KUKA KRL program: EPS_2_25618_SANMH09_A_20250918115516.src

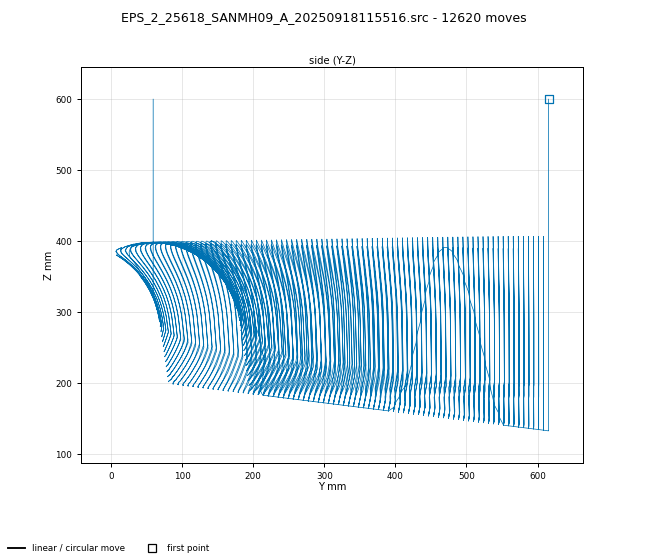
[picture p0: tool path of EPS_2_25618_SANMH09_A_20250918115516.src, 12620 of 12622 moves have a stored position in this frame; points joined in program order, loops and branches not executed]
&ACCESS RVP
&REL 4
&COMMENT QRS 19112012
&PARAM EDITMASK = *
DEF PART()
EXT BAS (BAS_COMMAND :IN,REAL :IN )
INT I
BAS (#INITMOV,0 )

;KUKA QRS Post kuka4.cps  Date:22-06-2017 !

File_ID=2845

QRS_PRE_INIT()

;Init var - Until changes are made in qrs_pre_init
Outlet_Square_prg=0
Inlet_1_Square_prg=0
Inlet_2_Square_prg=0
Inlet_3_Square_prg=0
Inlet_4_Square_prg=0
Inlet_5_Square_prg=0

Outlet_1={X 0.000, Y 546.330, Z 306.500, B 0.000, E1 0.000 }
Inlet_1={X 0.000, Y 547.540, Z 289.500, B 0.000, E1 144.000 }
Outlet_1_type=201
Inlet_1_type=201
;QRS#1=Sidecore dimensions
;QRS#2=200-8" PVC SDR 35
;QRS#3=200-8" PVC SDR 35
;QRS#4=
;QRS#5=
;QRS#6=
;QRS#7=
;QRS#8=
;QRS#9=12-08 PSX
;QRS#10=12-08 PSX
;QRS#11=
;QRS#12=
;QRS#13=
;QRS#14=
;QRS#15=
;QRS#16=1220x127x686 2,25'
;QRS#17=EPS Height
;QRS#18=407
;QRS#19=*
;QRS#20= UPDATED VERSION 22-06-2017
;QRS#21=*
Outlet_Square=0100
Inlet_1_Square=0100
Inlet_2_Square=0
Inlet_3_Square=0
Inlet_4_Square=0
Inlet_5_Square=0
Mill_Square=1
Outlet_Square_Prg=204
Inlet_1_Square_prg=204

QRS_INIT()

$ADVANCE=5

; T1
PTP {E1 173.601,E2 173.601}
PTP {X 0,Y 615.511,A -85,B 0,C 180,E1 173.601,E2 173.601,E3 0,E4 0,E5 0,E6 0}
QRS_SPEED_INIT()
LIN {X 0,Y 615.511,Z 600,A -85,B 0,C 180,E1 173.601,E2 173.601,E3 0,E4 0,E5 0,E6 0} C_VEL
LIN {X 0,Y 615.511,Z 143.374,A -85,B 0,C 180,E1 173.601,E2 173.601} C_VEL
LIN {X 0,Y 615.511,Z 135.2,A -85,B 0,C 180,E1 173.601,E2 173.601} C_VEL
LIN {X 0,Y 615.479,Z 133.2,A -85,B 0,C 180,E1 173.415,E2 173.415} C_VEL
LIN {X 0,Y 615.419,Z 133.199,A -85,B 0,C 180,E1 170.8,E2 170.8} C_VEL
LIN {X 0,Y 615.417,Z 133.199,A -85,B 0,C 180,E1 168.806,E2 168.806} C_VEL
LIN {X 0,Y 615.417,Z 133.199,A -85,B 0,C 180,E1 166.798,E2 166.798} C_VEL
LIN {X 0,Y 615.416,Z 133.199,A -85,B 0,C 180,E1 164.772,E2 164.772} C_VEL
LIN {X 0,Y 615.416,Z 133.199,A -85,B 0,C 180,E1 162.728,E2 162.728} C_VEL
LIN {X 0,Y 615.479,Z 133.198,A -85,B 0,C 180,E1 159.967,E2 159.967} C_VEL
LIN {X 0,Y 615.424,Z 133.199,A -85,B 0,C 180,E1 157.153,E2 157.153} C_VEL
LIN {X 0,Y 615.417,Z 133.199,A -85,B 0,C 180,E1 155.006,E2 155.006} C_VEL
LIN {X 0,Y 615.417,Z 133.199,A -85,B 0,C 180,E1 152.82,E2 152.82} C_VEL
LIN {X 0,Y 615.468,Z 133.198,A -85,B 0,C 180,E1 150.206,E2 150.206} C_VEL
LIN {X 0,Y 615.441,Z 133.199,A -85,B 0,C 180,E1 147.54,E2 147.54} C_VEL
LIN {X 0,Y 615.498,Z 133.423,A -85,B 0,C 180,E1 145.915,E2 145.915} C_VEL
LIN {X 0,Y 615.474,Z 149.74,A -85,B 0,C 180,E1 143.318,E2 143.318} C_VEL
LIN {X 0,Y 615.475,Z 167.201,A -85,B 0,C 180,E1 140.594,E2 140.594} C_VEL
LIN {X 0,Y 615.461,Z 178.625,A -85,B 0,C 180,E1 138.859,E2 138.859} C_VEL
LIN {X 0,Y 615.461,Z 179.533,A -85,B 0,C 180,E1 138.811,E2 138.811} C_VEL
LIN {X 0,Y 615.497,Z 286.075,A -85,B 0,C 180,E1 137.54,E2 137.54} C_VEL
LIN {X 0,Y 615.498,Z 298.937,A -85,B 0,C 180,E1 137.257,E2 137.257} C_VEL
LIN {X 0,Y 615.497,Z 311.305,A -85,B 0,C 180,E1 136.853,E2 136.853} C_VEL
LIN {X 0,Y 615.495,Z 322.152,A -85,B 0,C 180,E1 136.38,E2 136.38} C_VEL
LIN {X 0,Y 615.483,Z 333.44,A -85,B 0,C 180,E1 135.753,E2 135.753} C_VEL
LIN {X 0,Y 615.499,Z 343.297,A -85,B 0,C 180,E1 135.066,E2 135.066} C_VEL
LIN {X 0,Y 615.497,Z 352.917,A -85,B 0,C 180,E1 134.245,E2 134.245} C_VEL
LIN {X 0,Y 615.497,Z 360.762,A -85,B 0,C 180,E1 133.43,E2 133.43} C_VEL
LIN {X 0,Y 615.5,Z 367.975,A -85,B 0,C 180,E1 132.524,E2 132.524} C_VEL
LIN {X 0,Y 615.496,Z 374.697,A -85,B 0,C 180,E1 131.471,E2 131.471} C_VEL
LIN {X 0,Y 615.495,Z 380.268,A -85,B 0,C 180,E1 130.347,E2 130.347} C_VEL
LIN {X 0,Y 615.497,Z 383.832,A -85,B 0,C 180,E1 129.405,E2 129.405} C_VEL
LIN {X 0,Y 615.494,Z 387.343,A -85,B 0,C 180,E1 128.067,E2 128.067} C_VEL
LIN {X 0,Y 615.492,Z 388.944,A -85,B 0,C 180,E1 126.938,E2 126.938} C_VEL
LIN {X 0,Y 615.497,Z 389.366,A -85,B 0,C 180,E1 125.835,E2 125.835} C_VEL
LIN {X 0,Y 615.495,Z 388.646,A -85,B 0,C 180,E1 124.702,E2 124.702} C_VEL
LIN {X 0,Y 615.497,Z 386.676,A -85,B 0,C 180,E1 123.536,E2 123.536} C_VEL
LIN {X 0,Y 615.497,Z 383.277,A -85,B 0,C 180,E1 122.333,E2 122.333} C_VEL
LIN {X 0,Y 615.495,Z 379.504,A -85,B 0,C 180,E1 121.385,E2 121.385} C_VEL
LIN {X 0,Y 615.496,Z 374.193,A -85,B 0,C 180,E1 120.348,E2 120.348} C_VEL
LIN {X 0,Y 615.496,Z 368.113,A -85,B 0,C 180,E1 119.405,E2 119.405} C_VEL
LIN {X 0,Y 615.498,Z 360.52,A -85,B 0,C 180,E1 118.453,E2 118.453} C_VEL
LIN {X 0,Y 615.497,Z 351.617,A -85,B 0,C 180,E1 117.544,E2 117.544} C_VEL
LIN {X 0,Y 615.499,Z 342.011,A -85,B 0,C 180,E1 116.745,E2 116.745} C_VEL
LIN {X 0,Y 615.468,Z 330.621,A -85,B 0,C 180,E1 115.988,E2 115.988} C_VEL
LIN {X 0,Y 615.498,Z 318.396,A -85,B 0,C 180,E1 115.351,E2 115.351} C_VEL
LIN {X 0,Y 615.499,Z 305.635,A -85,B 0,C 180,E1 114.855,E2 114.855} C_VEL
LIN {X 0,Y 615.496,Z 292.499,A -85,B 0,C 180,E1 114.495,E2 114.495} C_VEL
LIN {X 0,Y 615.496,Z 280.724,A -85,B 0,C 180,E1 114.293,E2 114.293} C_VEL
LIN {X 0,Y 615.451,Z 179.253,A -85,B 0,C 180,E1 113.089,E2 113.089} C_VEL
LIN {X 0,Y 615.455,Z 178.329,A -85,B 0,C 180,E1 113.022,E2 113.022} C_VEL
LIN {X 0,Y 615.454,Z 160.623,A -85,B 0,C 180,E1 110.294,E2 110.294} C_VEL
LIN {X 0,Y 615.45,Z 144.623,A -85,B 0,C 180,E1 107.785,E2 107.785} C_VEL
LIN {X 0,Y 615.493,Z 133.34,A -85,B 0,C 180,E1 105.97,E2 105.97} C_VEL
LIN {X 0,Y 615.471,Z 133.187,A -85,B 0,C 180,E1 103.201,E2 103.201} C_VEL
LIN {X 0,Y 615.487,Z 133.188,A -85,B 0,C 180,E1 100.526,E2 100.526} C_VEL
LIN {X 0,Y 615.482,Z 133.197,A -85,B 0,C 180,E1 97.875,E2 97.875} C_VEL
LIN {X 0,Y 615.474,Z 133.186,A -85,B 0,C 180,E1 95.241,E2 95.241} C_VEL
LIN {X 0,Y 615.487,Z 133.19,A -85,B 0,C 180,E1 92.617,E2 92.617} C_VEL
LIN {X 0,Y 615.477,Z 133.196,A -85,B 0,C 180,E1 89.999,E2 89.999} C_VEL
LIN {X 0,Y 615.472,Z 133.186,A -85,B 0,C 180,E1 87.381,E2 87.381} C_VEL
LIN {X 0,Y 615.489,Z 133.19,A -85,B 0,C 180,E1 84.758,E2 84.758} C_VEL
LIN {X 0,Y 615.473,Z 133.196,A -85,B 0,C 180,E1 82.124,E2 82.124} C_VEL
LIN {X 0,Y 615.473,Z 133.186,A -85,B 0,C 180,E1 79.472,E2 79.472} C_VEL
LIN {X 0,Y 615.49,Z 133.193,A -85,B 0,C 180,E1 76.798,E2 76.798} C_VEL
LIN {X 0,Y 615.462,Z 133.193,A -85,B 0,C 180,E1 74.094,E2 74.094} C_VEL
LIN {X 0,Y 615.486,Z 133.185,A -85,B 0,C 180,E1 71.354,E2 71.354} C_VEL
LIN {X 0,Y 615.483,Z 133.198,A -85,B 0,C 180,E1 68.568,E2 68.568} C_VEL
LIN {X 0,Y 615.458,Z 133.19,A -85,B 0,C 180,E1 65.997,E2 65.997} C_VEL
LIN {X 0,Y 615.482,Z 133.185,A -85,B 0,C 180,E1 63.555,E2 63.555} C_VEL
LIN {X 0,Y 615.47,Z 133.197,A -85,B 0,C 180,E1 60.593,E2 60.593} C_VEL
LIN {X 0,Y 615.456,Z 133.193,A -85,B 0,C 180,E1 58.313,E2 58.313} C_VEL
LIN {X 0,Y 615.461,Z 133.189,A -85,B 0,C 180,E1 55.976,E2 55.976} C_VEL
LIN {X 0,Y 615.487,Z 133.203,A -85,B 0,C 180,E1 53.063,E2 53.063} C_VEL
LIN {X 0,Y 615.454,Z 133.191,A -85,B 0,C 180,E1 50.247,E2 50.247} C_VEL
LIN {X 0,Y 615.498,Z 133.186,A -85,B 0,C 180,E1 47.648,E2 47.648} C_VEL
LIN {X 0,Y 615.468,Z 133.197,A -85,B 0,C 180,E1 44.93,E2 44.93} C_VEL
LIN {X 0,Y 615.453,Z 133.191,A -85,B 0,C 180,E1 42.355,E2 42.355} C_VEL
LIN {X 0,Y 615.494,Z 133.189,A -85,B 0,C 180,E1 39.749,E2 39.749} C_VEL
LIN {X 0,Y 615.453,Z 133.196,A -85,B 0,C 180,E1 36.932,E2 36.932} C_VEL
LIN {X 0,Y 615.447,Z 133.193,A -85,B 0,C 180,E1 34.695,E2 34.695} C_VEL
LIN {X 0,Y 615.46,Z 133.19,A -85,B 0,C 180,E1 32.327,E2 32.327} C_VEL
LIN {X 0,Y 615.479,Z 133.199,A -85,B 0,C 180,E1 29.406,E2 29.406} C_VEL
LIN {X 0,Y 615.447,Z 133.195,A -85,B 0,C 180,E1 27.038,E2 27.038} C_VEL
LIN {X 0,Y 615.445,Z 133.194,A -85,B 0,C 180,E1 24.993,E2 24.993} C_VEL
LIN {X 0,Y 615.469,Z 133.19,A -85,B 0,C 180,E1 22.342,E2 22.342} C_VEL
LIN {X 0,Y 615.453,Z 133.197,A -85,B 0,C 180,E1 19.339,E2 19.339} C_VEL
LIN {X 0,Y 615.446,Z 133.196,A -85,B 0,C 180,E1 17.271,E2 17.271} C_VEL
LIN {X 0,Y 615.442,Z 133.195,A -85,B 0,C 180,E1 15.227,E2 15.227} C_VEL
LIN {X 0,Y 615.44,Z 133.195,A -85,B 0,C 180,E1 13.202,E2 13.202} C_VEL
LIN {X 0,Y 615.474,Z 133.19,A -85,B 0,C 180,E1 10.527,E2 10.527} C_VEL
LIN {X 0,Y 615.478,Z 133.199,A -85,B 0,C 180,E1 7.875,E2 7.875} C_VEL
LIN {X 0,Y 615.436,Z 133.195,A -85,B 0,C 180,E1 5.241,E2 5.241} C_VEL
LIN {X 0,Y 615.478,Z 133.191,A -85,B 0,C 180,E1 2.618,E2 2.618} C_VEL
LIN {X 0,Y 615.471,Z 133.199,A -85,B 0,C 180,E1 0,E2 0} C_VEL
LIN {X 0,Y 615.431,Z 133.196,A -85,B 0,C 180,E1 -2.618,E2 -2.618} C_VEL
LIN {X 0,Y 615.476,Z 133.192,A -85,B 0,C 180,E1 -5.242,E2 -5.242} C_VEL
LIN {X 0,Y 615.465,Z 133.199,A -85,B 0,C 180,E1 -7.876,E2 -7.876} C_VEL
LIN {X 0,Y 615.431,Z 133.196,A -85,B 0,C 180,E1 -10.528,E2 -10.528} C_VEL
LIN {X 0,Y 615.489,Z 133.193,A -85,B 0,C 180,E1 -13.201,E2 -13.201} C_VEL
LIN {X 0,Y 615.444,Z 133.198,A -85,B 0,C 180,E1 -15.907,E2 -15.907} C_VEL
LIN {X 0,Y 615.437,Z 133.198,A -85,B 0,C 180,E1 -17.959,E2 -17.959} C_VEL
LIN {X 0,Y 615.431,Z 133.198,A -85,B 0,C 180,E1 -20.035,E2 -20.035} C_VEL
LIN {X 0,Y 615.426,Z 133.197,A -85,B 0,C 180,E1 -22.332,E2 -22.332} C_VEL
LIN {X 0,Y 615.486,Z 133.194,A -85,B 0,C 180,E1 -24.992,E2 -24.992} C_VEL
LIN {X 0,Y 615.487,Z 133.202,A -85,B 0,C 180,E1 -27.177,E2 -27.177} C_VEL
LIN {X 0,Y 615.429,Z 133.198,A -85,B 0,C 180,E1 -29.785,E2 -29.785} C_VEL
LIN {X 0,Y 615.431,Z 133.199,A -85,B 0,C 180,E1 -31.689,E2 -31.689} C_VEL
LIN {X 0,Y 615.42,Z 133.198,A -85,B 0,C 180,E1 -34.027,E2 -34.027} C_VEL
LIN {X 0,Y 615.44,Z 133.197,A -85,B 0,C 180,E1 -36.428,E2 -36.428} C_VEL
LIN {X 0,Y 615.48,Z 133.2,A -85,B 0,C 180,E1 -39.061,E2 -39.061} C_VEL
LIN {X 0,Y 615.428,Z 133.199,A -85,B 0,C 180,E1 -41.479,E2 -41.479} C_VEL
LIN {X 0,Y 615.419,Z 133.199,A -85,B 0,C 180,E1 -43.991,E2 -43.991} C_VEL
LIN {X 0,Y 615.499,Z 133.2,A -85,B 0,C 180,E1 -46.756,E2 -46.756} C_VEL
LIN {X 0,Y 615.421,Z 133.2,A -85,B 0,C 180,E1 -49.388,E2 -49.388} C_VEL
LIN {X 0,Y 615.422,Z 133.2,A -85,B 0,C 180,E1 -51.996,E2 -51.996} C_VEL
LIN {X 0,Y 615.467,Z 133.2,A -85,B 0,C 180,E1 -54.383,E2 -54.383} C_VEL
LIN {X 0,Y 615.467,Z 133.2,A -85,B 0,C 180,E1 -56.762,E2 -56.762} C_VEL
LIN {X 0,Y 615.429,Z 133.2,A -85,B 0,C 180,E1 -59.077,E2 -59.077} C_VEL
LIN {X 0,Y 615.415,Z 133.199,A -85,B 0,C 180,E1 -61.338,E2 -61.338} C_VEL
LIN {X 0,Y 615.416,Z 133.199,A -85,B 0,C 180,E1 -63.552,E2 -63.552} C_VEL
LIN {X 0,Y 615.451,Z 133.2,A -85,B 0,C 180,E1 -66,E2 -66} C_VEL
LIN {X 0,Y 615.49,Z 133.315,A -85,B 0,C 180,E1 -68.348,E2 -68.348} C_VEL
LIN {X 0,Y 615.496,Z 136.92,A -85,B 0,C 180,E1 -68.919,E2 -68.919} C_VEL
LIN {X 0,Y 615.489,Z 156.474,A -85,B 0,C 180,E1 -71.722,E2 -71.722} C_VEL
LIN {X 0,Y 615.485,Z 176.888,A -85,B 0,C 180,E1 -74.604,E2 -74.604} C_VEL
LIN {X 0,Y 615.488,Z 194.896,A -85,B 0,C 180,E1 -77.092,E2 -77.092} C_VEL
LIN {X 0,Y 615.487,Z 196.853,A -85,B 0,C 180,E1 -77.155,E2 -77.155} C_VEL
LIN {X 0,Y 615.498,Z 302.799,A -85,B 0,C 180,E1 -78.41,E2 -78.41} C_VEL
LIN {X 0,Y 615.498,Z 315.323,A -85,B 0,C 180,E1 -78.682,E2 -78.682} C_VEL
LIN {X 0,Y 615.496,Z 328.504,A -85,B 0,C 180,E1 -79.109,E2 -79.109} C_VEL
LIN {X 0,Y 615.489,Z 340.466,A -85,B 0,C 180,E1 -79.639,E2 -79.639} C_VEL
LIN {X 0,Y 615.496,Z 351.985,A -85,B 0,C 180,E1 -80.303,E2 -80.303} C_VEL
LIN {X 0,Y 615.499,Z 362.334,A -85,B 0,C 180,E1 -81.049,E2 -81.049} C_VEL
LIN {X 0,Y 615.497,Z 370.806,A -85,B 0,C 180,E1 -81.794,E2 -81.794} C_VEL
LIN {X 0,Y 615.498,Z 378.601,A -85,B 0,C 180,E1 -82.619,E2 -82.619} C_VEL
LIN {X 0,Y 615.496,Z 386.199,A -85,B 0,C 180,E1 -83.607,E2 -83.607} C_VEL
LIN {X 0,Y 615.498,Z 393.201,A -85,B 0,C 180,E1 -84.758,E2 -84.758} C_VEL
LIN {X 0,Y 615.494,Z 397.849,A -85,B 0,C 180,E1 -85.743,E2 -85.743} C_VEL
LIN {X 0,Y 615.494,Z 401.397,A -85,B 0,C 180,E1 -86.726,E2 -86.726} C_VEL
LIN {X 0,Y 615.497,Z 403.231,A -85,B 0,C 180,E1 -87.382,E2 -87.382} C_VEL
LIN {X 0,Y 615.5,Z 404.606,A -85,B 0,C 180,E1 -88.036,E2 -88.036} C_VEL
LIN {X 0,Y 615.496,Z 406.173,A -85,B 0,C 180,E1 -89.345,E2 -89.345} C_VEL
LIN {X 0,Y 615.494,Z 406.389,A -85,B 0,C 180,E1 -89.999,E2 -89.999} C_VEL
LIN {X 0,Y 615.495,Z 405.581,A -85,B 0,C 180,E1 -91.308,E2 -91.308} C_VEL
LIN {X 0,Y 615.5,Z 404.609,A -85,B 0,C 180,E1 -91.962,E2 -91.962} C_VEL
LIN {X 0,Y 615.497,Z 403.235,A -85,B 0,C 180,E1 -92.617,E2 -92.617} C_VEL
LIN {X 0,Y 615.496,Z 400.352,A -85,B 0,C 180,E1 -93.6,E2 -93.6} C_VEL
LIN {X 0,Y 615.498,Z 396.445,A -85,B 0,C 180,E1 -94.584,E2 -94.584} C_VEL
LIN {X 0,Y 615.499,Z 391.409,A -85,B 0,C 180,E1 -95.569,E2 -95.569} C_VEL
LIN {X 0,Y 615.497,Z 384.87,A -85,B 0,C 180,E1 -96.583,E2 -96.583} C_VEL
LIN {X 0,Y 615.497,Z 377.14,A -85,B 0,C 180,E1 -97.545,E2 -97.545} C_VEL
LIN {X 0,Y 615.498,Z 369.054,A -85,B 0,C 180,E1 -98.37,E2 -98.37} C_VEL
LIN {X 0,Y 615.499,Z 359.178,A -85,B 0,C 180,E1 -99.198,E2 -99.198} C_VEL
LIN {X 0,Y 615.494,Z 347.995,A -85,B 0,C 180,E1 -99.944,E2 -99.944} C_VEL
LIN {X 0,Y 615.492,Z 337.039,A -85,B 0,C 180,E1 -100.526,E2 -100.526} C_VEL
LIN {X 0,Y 615.499,Z 324.43,A -85,B 0,C 180,E1 -101.042,E2 -101.042} C_VEL
LIN {X 0,Y 615.499,Z 312.101,A -85,B 0,C 180,E1 -101.4,E2 -101.4} C_VEL
LIN {X 0,Y 615.499,Z 298.526,A -85,B 0,C 180,E1 -101.651,E2 -101.651} C_VEL
LIN {X 0,Y 615.487,Z 195.739,A -85,B 0,C 180,E1 -102.865,E2 -102.865} C_VEL
LIN {X 0,Y 615.486,Z 194.486,A -85,B 0,C 180,E1 -102.948,E2 -102.948} C_VEL
LIN {X 0,Y 615.496,Z 173.267,A -85,B 0,C 180,E1 -105.904,E2 -105.904} C_VEL
LIN {X 0,Y 615.473,Z 153.898,A -85,B 0,C 180,E1 -108.645,E2 -108.645} C_VEL
LIN {X 0,Y 615.498,Z 134.505,A -85,B 0,C 180,E1 -111.43,E2 -111.43} C_VEL
LIN {X 0,Y 615.491,Z 133.318,A -85,B 0,C 180,E1 -111.65,E2 -111.65} C_VEL
LIN {X 0,Y 615.427,Z 133.199,A -85,B 0,C 180,E1 -114.273,E2 -114.273} C_VEL
LIN {X 0,Y 615.418,Z 133.199,A -85,B 0,C 180,E1 -116.446,E2 -116.446} C_VEL
LIN {X 0,Y 615.417,Z 133.199,A -85,B 0,C 180,E1 -118.66,E2 -118.66} C_VEL
LIN {X 0,Y 615.445,Z 133.198,A -85,B 0,C 180,E1 -121.079,E2 -121.079} C_VEL
LIN {X 0,Y 615.434,Z 133.199,A -85,B 0,C 180,E1 -124.024,E2 -124.024} C_VEL
LIN {X 0,Y 615.416,Z 133.199,A -85,B 0,C 180,E1 -126.428,E2 -126.428} C_VEL
LIN {X 0,Y 615.457,Z 133.198,A -85,B 0,C 180,E1 -129.058,E2 -129.058} C_VEL
LIN {X 0,Y 615.484,Z 133.2,A -85,B 0,C 180,E1 -131.472,E2 -131.472} C_VEL
LIN {X 0,Y 615.424,Z 133.199,A -85,B 0,C 180,E1 -133.991,E2 -133.991} C_VEL
LIN {X 0,Y 615.422,Z 133.199,A -85,B 0,C 180,E1 -136.007,E2 -136.007} C_VEL
LIN {X 0,Y 615.459,Z 133.198,A -85,B 0,C 180,E1 -138.907,E2 -138.907} C_VEL
LIN {X 0,Y 615.482,Z 133.2,A -85,B 0,C 180,E1 -141.095,E2 -141.095} C_VEL
LIN {X 0,Y 615.445,Z 133.199,A -85,B 0,C 180,E1 -143.572,E2 -143.572} C_VEL
LIN {X 0,Y 615.417,Z 133.199,A -85,B 0,C 180,E1 -145.973,E2 -145.973} C_VEL
LIN {X 0,Y 615.468,Z 133.201,A -85,B 0,C 180,E1 -148.914,E2 -148.914} C_VEL
LIN {X 0,Y 615.434,Z 133.199,A -85,B 0,C 180,E1 -151.556,E2 -151.556} C_VEL
LIN {X 0,Y 615.43,Z 133.2,A -85,B 0,C 180,E1 -153.553,E2 -153.553} C_VEL
LIN {X 0,Y 615.42,Z 133.199,A -85,B 0,C 180,E1 -155.725,E2 -155.725} C_VEL
LIN {X 0,Y 615.414,Z 133.199,A -85,B 0,C 180,E1 -157.86,E2 -157.86} C_VEL
LIN {X 0,Y 615.475,Z 133.198,A -85,B 0,C 180,E1 -160.661,E2 -160.661} C_VEL
LIN {X 0,Y 615.43,Z 133.199,A -85,B 0,C 180,E1 -163.411,E2 -163.411} C_VEL
LIN {X 0,Y 615.425,Z 133.199,A -85,B 0,C 180,E1 -165.449,E2 -165.449} C_VEL
LIN {X 0,Y 615.421,Z 133.2,A -85,B 0,C 180,E1 -167.468,E2 -167.468} C_VEL
LIN {X 0,Y 615.421,Z 133.199,A -85,B 0,C 180,E1 -169.472,E2 -169.472} C_VEL
LIN {X 0,Y 615.42,Z 133.199,A -85,B 0,C 180,E1 -171.462,E2 -171.462} C_VEL
LIN {X 0,Y 615.419,Z 133.199,A -85,B 0,C 180,E1 -173.464,E2 -173.464} C_VEL
LIN {X 0,Y 615.419,Z 133.199,A -85,B 0,C 180,E1 -175.415,E2 -175.415} C_VEL
LIN {X 0,Y 615.419,Z 133.199,A -85,B 0,C 180,E1 -177.382,E2 -177.382} C_VEL
LIN {X 0,Y 615.419,Z 133.199,A -85,B 0,C 180,E1 -179.345,E2 -179.345} C_VEL
LIN {X 0,Y 615.419,Z 133.199,A -85,B 0,C 180,E1 -181.308,E2 -181.308} C_VEL
LIN {X 0,Y 615.42,Z 133.199,A -85,B 0,C 180,E1 -183.273,E2 -183.273} C_VEL
LIN {X 0,Y 615.419,Z 133.199,A -85,B 0,C 180,E1 -185.241,E2 -185.241} C_VEL
LIN {X 0,Y 615.479,Z 133.2,A -85,B 0,C 180,E1 -186.585,E2 -186.585} C_VEL
LIN {X 0,Y 614.762,Z 133.343,A -85,B 0,C 180,E1 -187.131,E2 -187.131} C_VEL
LIN {X 0,Y 611.898,Z 133.762,A -85,B 0,C 180,E1 -188.016,E2 -188.016} C_VEL
LIN {X 0,Y 609.51,Z 134.068,A -85,B 0,C 180,E1 -188.729,E2 -188.729} C_VEL
LIN {X 0,Y 608.487,Z 134.184,A -85,B 0,C 180,E1 -189.278,E2 -189.278} C_VEL
LIN {X 0,Y 608.404,Z 134.193,A -85,B 0,C 180,E1 -189.464,E2 -189.464} C_VEL
LIN {X 0,Y 608.425,Z 134.195,A -85,B 0,C 180,E1 -192,E2 -192} C_VEL
LIN {X 0,Y 608.415,Z 134.196,A -85,B 0,C 180,E1 -194.722,E2 -194.722} C_VEL
LIN {X 0,Y 608.411,Z 134.195,A -85,B 0,C 180,E1 -196.785,E2 -196.785} C_VEL
LIN {X 0,Y 608.407,Z 134.194,A -85,B 0,C 180,E1 -199.572,E2 -199.572} C_VEL
LIN {X 0,Y 608.444,Z 134.194,A -85,B 0,C 180,E1 -202.477,E2 -202.477} C_VEL
LIN {X 0,Y 608.422,Z 134.195,A -85,B 0,C 180,E1 -204.572,E2 -204.572} C_VEL
LIN {X 0,Y 608.399,Z 134.194,A -85,B 0,C 180,E1 -207.196,E2 -207.196} C_VEL
LIN {X 0,Y 608.455,Z 134.196,A -85,B 0,C 180,E1 -209.972,E2 -209.972} C_VEL
LIN {X 0,Y 608.408,Z 134.193,A -85,B 0,C 180,E1 -212.882,E2 -212.882} C_VEL
LIN {X 0,Y 608.503,Z 134.36,A -85,B 0,C 180,E1 -213.991,E2 -213.991} C_VEL
LIN {X 0,Y 608.485,Z 149.959,A -85,B 0,C 180,E1 -216.5,E2 -216.5} C_VEL
LIN {X 0,Y 608.469,Z 167.747,A -85,B 0,C 180,E1 -219.3,E2 -219.3} C_VEL
LIN {X 0,Y 608.457,Z 178.957,A -85,B 0,C 180,E1 -221.011,E2 -221.011} C_VEL
LIN {X 0,Y 608.551,Z 181.657,A -85,B 0,C 180,E1 -221.072,E2 -221.072} C_VEL
LIN {X 0,Y 608.556,Z 286.362,A -85,B 0,C 180,E1 -222.329,E2 -222.329} C_VEL
LIN {X 0,Y 608.548,Z 299.877,A -85,B 0,C 180,E1 -222.636,E2 -222.636} C_VEL
LIN {X 0,Y 608.535,Z 311.966,A -85,B 0,C 180,E1 -223.041,E2 -223.041} C_VEL
LIN {X 0,Y 608.518,Z 323.48,A -85,B 0,C 180,E1 -223.556,E2 -223.556} C_VEL
LIN {X 0,Y 608.471,Z 334.774,A -85,B 0,C 180,E1 -224.208,E2 -224.208} C_VEL
LIN {X 0,Y 608.491,Z 345.723,A -85,B 0,C 180,E1 -225.001,E2 -225.001} C_VEL
LIN {X 0,Y 608.486,Z 354.61,A -85,B 0,C 180,E1 -225.792,E2 -225.792} C_VEL
LIN {X 0,Y 608.463,Z 362.891,A -85,B 0,C 180,E1 -226.691,E2 -226.691} C_VEL
LIN {X 0,Y 608.461,Z 370.2,A -85,B 0,C 180,E1 -227.665,E2 -227.665} C_VEL
LIN {X 0,Y 608.431,Z 377.116,A -85,B 0,C 180,E1 -228.823,E2 -228.823} C_VEL
LIN {X 0,Y 608.441,Z 381.192,A -85,B 0,C 180,E1 -229.697,E2 -229.697} C_VEL
LIN {X 0,Y 608.425,Z 384.869,A -85,B 0,C 180,E1 -230.707,E2 -230.707} C_VEL
LIN {X 0,Y 608.416,Z 387.619,A -85,B 0,C 180,E1 -231.765,E2 -231.765} C_VEL
LIN {X 0,Y 608.428,Z 389.574,A -85,B 0,C 180,E1 -233.085,E2 -233.085} C_VEL
LIN {X 0,Y 608.418,Z 389.986,A -85,B 0,C 180,E1 -233.958,E2 -233.958} C_VEL
LIN {X 0,Y 608.422,Z 389.499,A -85,B 0,C 180,E1 -235.098,E2 -235.098} C_VEL
LIN {X 0,Y 608.436,Z 387.61,A -85,B 0,C 180,E1 -236.329,E2 -236.329} C_VEL
LIN {X 0,Y 608.425,Z 384.551,A -85,B 0,C 180,E1 -237.482,E2 -237.482} C_VEL
LIN {X 0,Y 608.448,Z 379.734,A -85,B 0,C 180,E1 -238.732,E2 -238.732} C_VEL
LIN {X 0,Y 608.444,Z 374.312,A -85,B 0,C 180,E1 -239.774,E2 -239.774} C_VEL
LIN {X 0,Y 608.442,Z 367.632,A -85,B 0,C 180,E1 -240.791,E2 -240.791} C_VEL
LIN {X 0,Y 608.452,Z 359.971,A -85,B 0,C 180,E1 -241.735,E2 -241.735} C_VEL
LIN {X 0,Y 608.478,Z 350.611,A -85,B 0,C 180,E1 -242.674,E2 -242.674} C_VEL
LIN {X 0,Y 608.483,Z 340.259,A -85,B 0,C 180,E1 -243.506,E2 -243.506} C_VEL
LIN {X 0,Y 608.472,Z 330.233,A -85,B 0,C 180,E1 -244.162,E2 -244.162} C_VEL
LIN {X 0,Y 608.518,Z 318.045,A -85,B 0,C 180,E1 -244.795,E2 -244.795} C_VEL
LIN {X 0,Y 608.545,Z 306.43,A -85,B 0,C 180,E1 -245.252,E2 -245.252} C_VEL
LIN {X 0,Y 608.551,Z 292.698,A -85,B 0,C 180,E1 -245.636,E2 -245.636} C_VEL
LIN {X 0,Y 608.561,Z 279.311,A -85,B 0,C 180,E1 -245.862,E2 -245.862} C_VEL
LIN {X 0,Y 608.479,Z 179.332,A -85,B 0,C 180,E1 -247.058,E2 -247.058} C_VEL
LIN {X 0,Y 608.449,Z 177.72,A -85,B 0,C 180,E1 -247.237,E2 -247.237} C_VEL
LIN {X 0,Y 608.439,Z 159.539,A -85,B 0,C 180,E1 -250.078,E2 -250.078} C_VEL
LIN {X 0,Y 608.483,Z 144.079,A -85,B 0,C 180,E1 -252.525,E2 -252.525} C_VEL
LIN {X 0,Y 608.487,Z 134.291,A -85,B 0,C 180,E1 -254.123,E2 -254.123} C_VEL
LIN {X 0,Y 608.454,Z 134.189,A -85,B 0,C 180,E1 -256.644,E2 -256.644} C_VEL
LIN {X 0,Y 608.465,Z 134.188,A -85,B 0,C 180,E1 -259.351,E2 -259.351} C_VEL
LIN {X 0,Y 608.474,Z 134.193,A -85,B 0,C 180,E1 -262.034,E2 -262.034} C_VEL
LIN {X 0,Y 608.454,Z 134.188,A -85,B 0,C 180,E1 -264.699,E2 -264.699} C_VEL
LIN {X 0,Y 608.477,Z 134.188,A -85,B 0,C 180,E1 -267.353,E2 -267.353} C_VEL
LIN {X 0,Y 608.469,Z 134.192,A -85,B 0,C 180,E1 -270.001,E2 -270.001} C_VEL
LIN {X 0,Y 608.465,Z 134.186,A -85,B 0,C 180,E1 -272.649,E2 -272.649} C_VEL
LIN {X 0,Y 608.466,Z 134.191,A -85,B 0,C 180,E1 -275.302,E2 -275.302} C_VEL
LIN {X 0,Y 608.467,Z 134.19,A -85,B 0,C 180,E1 -277.968,E2 -277.968} C_VEL
LIN {X 0,Y 608.458,Z 134.187,A -85,B 0,C 180,E1 -280.65,E2 -280.65} C_VEL
LIN {X 0,Y 608.462,Z 134.195,A -85,B 0,C 180,E1 -283.357,E2 -283.357} C_VEL
LIN {X 0,Y 608.442,Z 134.19,A -85,B 0,C 180,E1 -286.095,E2 -286.095} C_VEL
LIN {X 0,Y 608.455,Z 134.19,A -85,B 0,C 180,E1 -288.87,E2 -288.87} C_VEL
LIN {X 0,Y 608.458,Z 134.191,A -85,B 0,C 180,E1 -291.692,E2 -291.692} C_VEL
LIN {X 0,Y 608.448,Z 134.189,A -85,B 0,C 180,E1 -294.572,E2 -294.572} C_VEL
LIN {X 0,Y 608.438,Z 134.194,A -85,B 0,C 180,E1 -297.519,E2 -297.519} C_VEL
LIN {X 0,Y 608.442,Z 134.189,A -85,B 0,C 180,E1 -299.968,E2 -299.968} C_VEL
LIN {X 0,Y 608.454,Z 134.195,A -85,B 0,C 180,E1 -302.88,E2 -302.88} C_VEL
LIN {X 0,Y 608.428,Z 134.196,A -85,B 0,C 180,E1 -305.279,E2 -305.279} C_VEL
LIN {X 0,Y 608.452,Z 134.188,A -85,B 0,C 180,E1 -307.748,E2 -307.748} C_VEL
LIN {X 0,Y 608.446,Z 134.191,A -85,B 0,C 180,E1 -310.329,E2 -310.329} C_VEL
LIN {X 0,Y 608.441,Z 134.197,A -85,B 0,C 180,E1 -312.961,E2 -312.961} C_VEL
LIN {X 0,Y 608.434,Z 134.19,A -85,B 0,C 180,E1 -315.738,E2 -315.738} C_VEL
LIN {X 0,Y 608.449,Z 134.188,A -85,B 0,C 180,E1 -317.938,E2 -317.938} C_VEL
LIN {X 0,Y 608.439,Z 134.199,A -85,B 0,C 180,E1 -320.706,E2 -320.706} C_VEL
LIN {X 0,Y 608.424,Z 134.194,A -85,B 0,C 180,E1 -323.083,E2 -323.083} C_VEL
LIN {X 0,Y 608.444,Z 134.188,A -85,B 0,C 180,E1 -325.53,E2 -325.53} C_VEL
LIN {X 0,Y 608.454,Z 134.189,A -85,B 0,C 180,E1 -327.905,E2 -327.905} C_VEL
LIN {X 0,Y 608.479,Z 134.191,A -85,B 0,C 180,E1 -330.221,E2 -330.221} C_VEL
LIN {X 0,Y 608.415,Z 134.192,A -85,B 0,C 180,E1 -333.225,E2 -333.225} C_VEL
LIN {X 0,Y 608.482,Z 134.187,A -85,B 0,C 180,E1 -335.846,E2 -335.846} C_VEL
LIN {X 0,Y 608.456,Z 134.197,A -85,B 0,C 180,E1 -338.308,E2 -338.308} C_VEL
LIN {X 0,Y 608.435,Z 134.19,A -85,B 0,C 180,E1 -341.13,E2 -341.13} C_VEL
LIN {X 0,Y 608.458,Z 134.193,A -85,B 0,C 180,E1 -343.906,E2 -343.906} C_VEL
LIN {X 0,Y 608.432,Z 134.192,A -85,B 0,C 180,E1 -346.643,E2 -346.643} C_VEL
LIN {X 0,Y 608.443,Z 134.19,A -85,B 0,C 180,E1 -349.35,E2 -349.35} C_VEL
LIN {X 0,Y 608.47,Z 134.195,A -85,B 0,C 180,E1 -352.033,E2 -352.033} C_VEL
LIN {X 0,Y 608.422,Z 134.192,A -85,B 0,C 180,E1 -354.698,E2 -354.698} C_VEL
LIN {X 0,Y 608.468,Z 134.188,A -85,B 0,C 180,E1 -357.352,E2 -357.352} C_VEL
LIN {X 0,Y 608.463,Z 134.193,A -85,B 0,C 180,E1 -360,E2 -360} C_VEL
LIN {X 0,Y 608.428,Z 134.191,A -85,B 0,C 180,E1 -362.649,E2 -362.649} C_VEL
LIN {X 0,Y 608.455,Z 134.191,A -85,B 0,C 180,E1 -365.302,E2 -365.302} C_VEL
LIN {X 0,Y 608.426,Z 134.195,A -85,B 0,C 180,E1 -367.968,E2 -367.968} C_VEL
LIN {X 0,Y 608.428,Z 134.194,A -85,B 0,C 180,E1 -369.978,E2 -369.978} C_VEL
LIN {X 0,Y 608.411,Z 134.193,A -85,B 0,C 180,E1 -372.679,E2 -372.679} C_VEL
LIN {X 0,Y 608.459,Z 134.197,A -85,B 0,C 180,E1 -375.407,E2 -375.407} C_VEL
LIN {X 0,Y 608.399,Z 134.195,A -85,B 0,C 180,E1 -378.174,E2 -378.174} C_VEL
LIN {X 0,Y 608.429,Z 134.192,A -85,B 0,C 180,E1 -380.669,E2 -380.669} C_VEL
LIN {X 0,Y 608.429,Z 134.198,A -85,B 0,C 180,E1 -383.125,E2 -383.125} C_VEL
LIN {X 0,Y 608.418,Z 134.195,A -85,B 0,C 180,E1 -385.711,E2 -385.711} C_VEL
LIN {X 0,Y 608.427,Z 134.196,A -85,B 0,C 180,E1 -387.519,E2 -387.519} C_VEL
LIN {X 0,Y 608.397,Z 134.195,A -85,B 0,C 180,E1 -389.96,E2 -389.96} C_VEL
LIN {X 0,Y 608.42,Z 134.194,A -85,B 0,C 180,E1 -392.516,E2 -392.516} C_VEL
LIN {X 0,Y 608.412,Z 134.198,A -85,B 0,C 180,E1 -395.28,E2 -395.28} C_VEL
LIN {X 0,Y 608.4,Z 134.194,A -85,B 0,C 180,E1 -397.752,E2 -397.752} C_VEL
LIN {X 0,Y 608.405,Z 134.195,A -85,B 0,C 180,E1 -400.324,E2 -400.324} C_VEL
LIN {X 0,Y 608.436,Z 134.193,A -85,B 0,C 180,E1 -403.305,E2 -403.305} C_VEL
LIN {X 0,Y 608.421,Z 134.193,A -85,B 0,C 180,E1 -406.126,E2 -406.126} C_VEL
LIN {X 0,Y 608.438,Z 134.198,A -85,B 0,C 180,E1 -408.822,E2 -408.822} C_VEL
LIN {X 0,Y 608.39,Z 134.196,A -85,B 0,C 180,E1 -411.406,E2 -411.406} C_VEL
LIN {X 0,Y 608.409,Z 134.196,A -85,B 0,C 180,E1 -413.082,E2 -413.082} C_VEL
LIN {X 0,Y 608.385,Z 134.196,A -85,B 0,C 180,E1 -415.525,E2 -415.525} C_VEL
LIN {X 0,Y 608.417,Z 134.193,A -85,B 0,C 180,E1 -417.902,E2 -417.902} C_VEL
LIN {X 0,Y 608.444,Z 134.195,A -85,B 0,C 180,E1 -420.219,E2 -420.219} C_VEL
LIN {X 0,Y 608.389,Z 134.196,A -85,B 0,C 180,E1 -423.223,E2 -423.223} C_VEL
LIN {X 0,Y 608.404,Z 134.194,A -85,B 0,C 180,E1 -425.426,E2 -425.426} C_VEL
LIN {X 0,Y 608.5,Z 134.353,A -85,B 0,C 180,E1 -428.265,E2 -428.265} C_VEL
LIN {X 0,Y 608.556,Z 149.064,A -85,B 0,C 180,E1 -430.432,E2 -430.432} C_VEL
LIN {X 0,Y 608.481,Z 168.482,A -85,B 0,C 180,E1 -433.216,E2 -433.216} C_VEL
LIN {X 0,Y 608.484,Z 188.014,A -85,B 0,C 180,E1 -435.978,E2 -435.978} C_VEL
LIN {X 0,Y 608.499,Z 195.248,A -85,B 0,C 180,E1 -436.962,E2 -436.962} C_VEL
LIN {X 0,Y 608.564,Z 200.465,A -85,B 0,C 180,E1 -437.049,E2 -437.049} C_VEL
LIN {X 0,Y 608.549,Z 302.918,A -85,B 0,C 180,E1 -438.276,E2 -438.276} C_VEL
LIN {X 0,Y 608.548,Z 316.197,A -85,B 0,C 180,E1 -438.572,E2 -438.572} C_VEL
LIN {X 0,Y 608.545,Z 329.328,A -85,B 0,C 180,E1 -439.009,E2 -439.009} C_VEL
LIN {X 0,Y 608.51,Z 340.624,A -85,B 0,C 180,E1 -439.519,E2 -439.519} C_VEL
LIN {X 0,Y 608.488,Z 352.189,A -85,B 0,C 180,E1 -440.191,E2 -440.191} C_VEL
LIN {X 0,Y 608.485,Z 362.587,A -85,B 0,C 180,E1 -440.945,E2 -440.945} C_VEL
LIN {X 0,Y 608.475,Z 371.106,A -85,B 0,C 180,E1 -441.698,E2 -441.698} C_VEL
LIN {X 0,Y 608.471,Z 378.955,A -85,B 0,C 180,E1 -442.533,E2 -442.533} C_VEL
LIN {X 0,Y 608.461,Z 386.285,A -85,B 0,C 180,E1 -443.484,E2 -443.484} C_VEL
LIN {X 0,Y 608.451,Z 391.862,A -85,B 0,C 180,E1 -444.365,E2 -444.365} C_VEL
LIN {X 0,Y 608.432,Z 396.947,A -85,B 0,C 180,E1 -445.362,E2 -445.362} C_VEL
LIN {X 0,Y 608.449,Z 400.894,A -85,B 0,C 180,E1 -446.357,E2 -446.357} C_VEL
LIN {X 0,Y 608.425,Z 403.807,A -85,B 0,C 180,E1 -447.351,E2 -447.351} C_VEL
LIN {X 0,Y 608.445,Z 405.2,A -85,B 0,C 180,E1 -448.014,E2 -448.014} C_VEL
LIN {X 0,Y 608.439,Z 406.783,A -85,B 0,C 180,E1 -449.337,E2 -449.337} C_VEL
LIN {X 0,Y 608.434,Z 407,A -85,B 0,C 180,E1 -449.999,E2 -449.999} C_VEL
LIN {X 0,Y 608.448,Z 406.185,A -85,B 0,C 180,E1 -451.323,E2 -451.323} C_VEL
LIN {X 0,Y 608.444,Z 405.203,A -85,B 0,C 180,E1 -451.985,E2 -451.985} C_VEL
LIN {X 0,Y 608.425,Z 403.811,A -85,B 0,C 180,E1 -452.648,E2 -452.648} C_VEL
LIN {X 0,Y 608.449,Z 400.899,A -85,B 0,C 180,E1 -453.642,E2 -453.642} C_VEL
LIN {X 0,Y 608.432,Z 396.953,A -85,B 0,C 180,E1 -454.637,E2 -454.637} C_VEL
LIN {X 0,Y 608.438,Z 390.881,A -85,B 0,C 180,E1 -455.8,E2 -455.8} C_VEL
LIN {X 0,Y 608.462,Z 384.241,A -85,B 0,C 180,E1 -456.799,E2 -456.799} C_VEL
LIN {X 0,Y 608.455,Z 375.996,A -85,B 0,C 180,E1 -457.799,E2 -457.799} C_VEL
LIN {X 0,Y 608.472,Z 367.546,A -85,B 0,C 180,E1 -458.635,E2 -458.635} C_VEL
LIN {X 0,Y 608.479,Z 357.103,A -85,B 0,C 180,E1 -459.473,E2 -459.473} C_VEL
LIN {X 0,Y 608.497,Z 346.77,A -85,B 0,C 180,E1 -460.144,E2 -460.144} C_VEL
LIN {X 0,Y 608.522,Z 335.254,A -85,B 0,C 180,E1 -460.74,E2 -460.74} C_VEL
LIN {X 0,Y 608.533,Z 323.895,A -85,B 0,C 180,E1 -461.192,E2 -461.192} C_VEL
LIN {X 0,Y 608.562,Z 310.391,A -85,B 0,C 180,E1 -461.574,E2 -461.574} C_VEL
LIN {X 0,Y 608.551,Z 297.152,A -85,B 0,C 180,E1 -461.807,E2 -461.807} C_VEL
LIN {X 0,Y 608.549,Z 195.747,A -85,B 0,C 180,E1 -463.014,E2 -463.014} C_VEL
LIN {X 0,Y 608.462,Z 194.617,A -85,B 0,C 180,E1 -463.101,E2 -463.101} C_VEL
LIN {X 0,Y 608.501,Z 174.56,A -85,B 0,C 180,E1 -465.92,E2 -465.92} C_VEL
LIN {X 0,Y 608.502,Z 156.515,A -85,B 0,C 180,E1 -468.495,E2 -468.495} C_VEL
LIN {X 0,Y 608.57,Z 138.151,A -85,B 0,C 180,E1 -471.154,E2 -471.154} C_VEL
LIN {X 0,Y 608.471,Z 134.299,A -85,B 0,C 180,E1 -471.757,E2 -471.757} C_VEL
LIN {X 0,Y 608.404,Z 134.194,A -85,B 0,C 180,E1 -474.572,E2 -474.572} C_VEL
LIN {X 0,Y 608.39,Z 134.195,A -85,B 0,C 180,E1 -476.776,E2 -476.776} C_VEL
LIN {X 0,Y 608.449,Z 134.195,A -85,B 0,C 180,E1 -479.779,E2 -479.779} C_VEL
LIN {X 0,Y 608.402,Z 134.194,A -85,B 0,C 180,E1 -482.513,E2 -482.513} C_VEL
LIN {X 0,Y 608.399,Z 134.196,A -85,B 0,C 180,E1 -484.898,E2 -484.898} C_VEL
LIN {X 0,Y 608.431,Z 134.195,A -85,B 0,C 180,E1 -487.747,E2 -487.747} C_VEL
LIN {X 0,Y 608.394,Z 134.195,A -85,B 0,C 180,E1 -490.322,E2 -490.322} C_VEL
LIN {X 0,Y 608.424,Z 134.195,A -85,B 0,C 180,E1 -492.961,E2 -492.961} C_VEL
LIN {X 0,Y 608.41,Z 134.196,A -85,B 0,C 180,E1 -495.739,E2 -495.739} C_VEL
LIN {X 0,Y 608.409,Z 134.194,A -85,B 0,C 180,E1 -497.934,E2 -497.934} C_VEL
LIN {X 0,Y 608.416,Z 134.195,A -85,B 0,C 180,E1 -500.707,E2 -500.707} C_VEL
LIN {X 0,Y 608.442,Z 134.198,A -85,B 0,C 180,E1 -503.084,E2 -503.084} C_VEL
LIN {X 0,Y 608.443,Z 134.193,A -85,B 0,C 180,E1 -505.529,E2 -505.529} C_VEL
LIN {X 0,Y 608.412,Z 134.193,A -85,B 0,C 180,E1 -507.902,E2 -507.902} C_VEL
LIN {X 0,Y 608.406,Z 134.193,A -85,B 0,C 180,E1 -510.217,E2 -510.217} C_VEL
LIN {X 0,Y 608.454,Z 134.194,A -85,B 0,C 180,E1 -512.794,E2 -512.794} C_VEL
LIN {X 0,Y 608.422,Z 134.195,A -85,B 0,C 180,E1 -515.427,E2 -515.427} C_VEL
LIN {X 0,Y 608.423,Z 134.193,A -85,B 0,C 180,E1 -518.306,E2 -518.306} C_VEL
LIN {X 0,Y 608.435,Z 134.193,A -85,B 0,C 180,E1 -521.289,E2 -521.289} C_VEL
LIN {X 0,Y 608.4,Z 134.194,A -85,B 0,C 180,E1 -523.904,E2 -523.904} C_VEL
LIN {X 0,Y 608.456,Z 134.195,A -85,B 0,C 180,E1 -526.643,E2 -526.643} C_VEL
LIN {X 0,Y 608.411,Z 134.194,A -85,B 0,C 180,E1 -529.349,E2 -529.349} C_VEL
LIN {X 0,Y 608.405,Z 134.195,A -85,B 0,C 180,E1 -531.363,E2 -531.363} C_VEL
LIN {X 0,Y 608.398,Z 134.195,A -85,B 0,C 180,E1 -533.421,E2 -533.421} C_VEL
LIN {X 0,Y 608.393,Z 134.196,A -85,B 0,C 180,E1 -535.362,E2 -535.362} C_VEL
LIN {X 0,Y 608.417,Z 134.192,A -85,B 0,C 180,E1 -537.351,E2 -537.351} C_VEL
LIN {X 0,Y 608.398,Z 134.195,A -85,B 0,C 180,E1 -539.338,E2 -539.338} C_VEL
LIN {X 0,Y 608.408,Z 134.193,A -85,B 0,C 180,E1 -541.324,E2 -541.324} C_VEL
LIN {X 0,Y 608.389,Z 134.196,A -85,B 0,C 180,E1 -543.311,E2 -543.311} C_VEL
LIN {X 0,Y 608.403,Z 134.194,A -85,B 0,C 180,E1 -545.302,E2 -545.302} C_VEL
LIN {X 0,Y 608.397,Z 134.195,A -85,B 0,C 180,E1 -547.3,E2 -547.3} C_VEL
LIN {X 0,Y 608.404,Z 134.193,A -85,B 0,C 180,E1 -549.464,E2 -549.464} C_VEL
LIN {X 0,Y 607.738,Z 134.282,A -85,B 0,C 180,E1 -550.017,E2 -550.017} C_VEL
LIN {X 0,Y 604.894,Z 134.637,A -85,B 0,C 180,E1 -550.914,E2 -550.914} C_VEL
LIN {X 0,Y 602.492,Z 134.937,A -85,B 0,C 180,E1 -551.636,E2 -551.636} C_VEL
LIN {X 0,Y 601.46,Z 135.066,A -85,B 0,C 180,E1 -552.192,E2 -552.192} C_VEL
LIN {X 0,Y 601.376,Z 135.073,A -85,B 0,C 180,E1 -552.381,E2 -552.381} C_VEL
LIN {X 0,Y 601.377,Z 135.071,A -85,B 0,C 180,E1 -554.898,E2 -554.898} C_VEL
LIN {X 0,Y 601.382,Z 135.069,A -85,B 0,C 180,E1 -556.987,E2 -556.987} C_VEL
LIN {X 0,Y 601.372,Z 135.073,A -85,B 0,C 180,E1 -559.81,E2 -559.81} C_VEL
LIN {X 0,Y 601.391,Z 135.07,A -85,B 0,C 180,E1 -562.683,E2 -562.683} C_VEL
LIN {X 0,Y 601.362,Z 135.071,A -85,B 0,C 180,E1 -564.88,E2 -564.88} C_VEL
LIN {X 0,Y 601.359,Z 135.072,A -85,B 0,C 180,E1 -567.355,E2 -567.355} C_VEL
LIN {X 0,Y 601.391,Z 135.077,A -85,B 0,C 180,E1 -570.166,E2 -570.166} C_VEL
LIN {X 0,Y 601.381,Z 135.07,A -85,B 0,C 180,E1 -572.712,E2 -572.712} C_VEL
LIN {X 0,Y 601.443,Z 135.257,A -85,B 0,C 180,E1 -573.894,E2 -573.894} C_VEL
LIN {X 0,Y 601.504,Z 148.217,A -85,B 0,C 180,E1 -576.009,E2 -576.009} C_VEL
LIN {X 0,Y 601.474,Z 165.495,A -85,B 0,C 180,E1 -578.767,E2 -578.767} C_VEL
LIN {X 0,Y 601.429,Z 178.875,A -85,B 0,C 180,E1 -580.851,E2 -580.851} C_VEL
LIN {X 0,Y 601.658,Z 181.849,A -85,B 0,C 180,E1 -580.923,E2 -580.923} C_VEL
LIN {X 0,Y 601.606,Z 286.775,A -85,B 0,C 180,E1 -582.199,E2 -582.199} C_VEL
LIN {X 0,Y 601.578,Z 300.522,A -85,B 0,C 180,E1 -582.52,E2 -582.52} C_VEL
LIN {X 0,Y 601.561,Z 312.735,A -85,B 0,C 180,E1 -582.942,E2 -582.942} C_VEL
LIN {X 0,Y 601.514,Z 325.132,A -85,B 0,C 180,E1 -583.522,E2 -583.522} C_VEL
LIN {X 0,Y 601.451,Z 335.85,A -85,B 0,C 180,E1 -584.164,E2 -584.164} C_VEL
LIN {X 0,Y 601.457,Z 345.75,A -85,B 0,C 180,E1 -584.897,E2 -584.897} C_VEL
LIN {X 0,Y 601.414,Z 354.835,A -85,B 0,C 180,E1 -585.717,E2 -585.717} C_VEL
LIN {X 0,Y 601.404,Z 363.31,A -85,B 0,C 180,E1 -586.656,E2 -586.656} C_VEL
LIN {X 0,Y 601.373,Z 370.397,A -85,B 0,C 180,E1 -587.619,E2 -587.619} C_VEL
LIN {X 0,Y 601.358,Z 377.136,A -85,B 0,C 180,E1 -588.767,E2 -588.767} C_VEL
LIN {X 0,Y 601.352,Z 382.598,A -85,B 0,C 180,E1 -590.002,E2 -590.002} C_VEL
LIN {X 0,Y 601.318,Z 385.488,A -85,B 0,C 180,E1 -590.868,E2 -590.868} C_VEL
LIN {X 0,Y 601.329,Z 387.59,A -85,B 0,C 180,E1 -591.727,E2 -591.727} C_VEL
LIN {X 0,Y 601.326,Z 389.095,A -85,B 0,C 180,E1 -592.631,E2 -592.631} C_VEL
LIN {X 0,Y 601.311,Z 389.938,A -85,B 0,C 180,E1 -593.751,E2 -593.751} C_VEL
LIN {X 0,Y 601.334,Z 389.54,A -85,B 0,C 180,E1 -595.064,E2 -595.064} C_VEL
LIN {X 0,Y 601.323,Z 388.163,A -85,B 0,C 180,E1 -596.079,E2 -596.079} C_VEL
LIN {X 0,Y 601.332,Z 385.254,A -85,B 0,C 180,E1 -597.297,E2 -597.297} C_VEL
LIN {X 0,Y 601.353,Z 381.902,A -85,B 0,C 180,E1 -598.272,E2 -598.272} C_VEL
LIN {X 0,Y 601.356,Z 376.489,A -85,B 0,C 180,E1 -599.445,E2 -599.445} C_VEL
LIN {X 0,Y 601.376,Z 369.501,A -85,B 0,C 180,E1 -600.606,E2 -600.606} C_VEL
LIN {X 0,Y 601.405,Z 362.258,A -85,B 0,C 180,E1 -601.564,E2 -601.564} C_VEL
LIN {X 0,Y 601.414,Z 352.916,A -85,B 0,C 180,E1 -602.557,E2 -602.557} C_VEL
LIN {X 0,Y 601.455,Z 342.497,A -85,B 0,C 180,E1 -603.453,E2 -603.453} C_VEL
LIN {X 0,Y 601.472,Z 331.397,A -85,B 0,C 180,E1 -604.21,E2 -604.21} C_VEL
LIN {X 0,Y 601.532,Z 319.489,A -85,B 0,C 180,E1 -604.851,E2 -604.851} C_VEL
LIN {X 0,Y 601.559,Z 307.99,A -85,B 0,C 180,E1 -605.329,E2 -605.329} C_VEL
LIN {X 0,Y 601.582,Z 294.964,A -85,B 0,C 180,E1 -605.719,E2 -605.719} C_VEL
LIN {X 0,Y 601.61,Z 282.354,A -85,B 0,C 180,E1 -605.959,E2 -605.959} C_VEL
LIN {X 0,Y 601.489,Z 179.664,A -85,B 0,C 180,E1 -607.201,E2 -607.201} C_VEL
LIN {X 0,Y 601.42,Z 178.648,A -85,B 0,C 180,E1 -607.261,E2 -607.261} C_VEL
LIN {X 0,Y 601.435,Z 160.027,A -85,B 0,C 180,E1 -610.193,E2 -610.193} C_VEL
LIN {X 0,Y 601.526,Z 143.485,A -85,B 0,C 180,E1 -612.843,E2 -612.843} C_VEL
LIN {X 0,Y 601.47,Z 135.26,A -85,B 0,C 180,E1 -614.194,E2 -614.194} C_VEL
LIN {X 0,Y 601.416,Z 135.065,A -85,B 0,C 180,E1 -617.173,E2 -617.173} C_VEL
LIN {X 0,Y 601.432,Z 135.072,A -85,B 0,C 180,E1 -619.906,E2 -619.906} C_VEL
LIN {X 0,Y 601.434,Z 135.063,A -85,B 0,C 180,E1 -622.616,E2 -622.616} C_VEL
LIN {X 0,Y 601.422,Z 135.066,A -85,B 0,C 180,E1 -625.309,E2 -625.309} C_VEL
LIN {X 0,Y 601.419,Z 135.071,A -85,B 0,C 180,E1 -627.992,E2 -627.992} C_VEL
LIN {X 0,Y 601.441,Z 135.061,A -85,B 0,C 180,E1 -630.67,E2 -630.67} C_VEL
LIN {X 0,Y 601.431,Z 135.067,A -85,B 0,C 180,E1 -633.35,E2 -633.35} C_VEL
LIN {X 0,Y 601.401,Z 135.07,A -85,B 0,C 180,E1 -636.038,E2 -636.038} C_VEL
LIN {X 0,Y 601.431,Z 135.065,A -85,B 0,C 180,E1 -638.061,E2 -638.061} C_VEL
LIN {X 0,Y 601.425,Z 135.066,A -85,B 0,C 180,E1 -641.014,E2 -641.014} C_VEL
LIN {X 0,Y 601.406,Z 135.075,A -85,B 0,C 180,E1 -643.517,E2 -643.517} C_VEL
LIN {X 0,Y 601.425,Z 135.063,A -85,B 0,C 180,E1 -646.288,E2 -646.288} C_VEL
LIN {X 0,Y 601.416,Z 135.07,A -85,B 0,C 180,E1 -649.099,E2 -649.099} C_VEL
LIN {X 0,Y 601.404,Z 135.075,A -85,B 0,C 180,E1 -651.24,E2 -651.24} C_VEL
LIN {X 0,Y 601.438,Z 135.061,A -85,B 0,C 180,E1 -654.142,E2 -654.142} C_VEL
LIN {X 0,Y 601.453,Z 135.069,A -85,B 0,C 180,E1 -657.111,E2 -657.111} C_VEL
LIN {X 0,Y 601.404,Z 135.071,A -85,B 0,C 180,E1 -659.394,E2 -659.394} C_VEL
LIN {X 0,Y 601.396,Z 135.068,A -85,B 0,C 180,E1 -661.728,E2 -661.728} C_VEL
LIN {X 0,Y 601.418,Z 135.064,A -85,B 0,C 180,E1 -664.119,E2 -664.119} C_VEL
LIN {X 0,Y 601.431,Z 135.065,A -85,B 0,C 180,E1 -667.382,E2 -667.382} C_VEL
LIN {X 0,Y 601.396,Z 135.067,A -85,B 0,C 180,E1 -669.996,E2 -669.996} C_VEL
LIN {X 0,Y 601.41,Z 135.073,A -85,B 0,C 180,E1 -672.671,E2 -672.671} C_VEL
LIN {X 0,Y 601.396,Z 135.067,A -85,B 0,C 180,E1 -675.48,E2 -675.48} C_VEL
LIN {X 0,Y 601.421,Z 135.069,A -85,B 0,C 180,E1 -678.407,E2 -678.407} C_VEL
LIN {X 0,Y 601.399,Z 135.072,A -85,B 0,C 180,E1 -680.873,E2 -680.873} C_VEL
LIN {X 0,Y 601.385,Z 135.068,A -85,B 0,C 180,E1 -683.416,E2 -683.416} C_VEL
LIN {X 0,Y 601.432,Z 135.065,A -85,B 0,C 180,E1 -686.064,E2 -686.064} C_VEL
LIN {X 0,Y 601.394,Z 135.068,A -85,B 0,C 180,E1 -689.057,E2 -689.057} C_VEL
LIN {X 0,Y 601.403,Z 135.066,A -85,B 0,C 180,E1 -691.372,E2 -691.372} C_VEL
LIN {X 0,Y 601.433,Z 135.072,A -85,B 0,C 180,E1 -694.383,E2 -694.383} C_VEL
LIN {X 0,Y 601.386,Z 135.073,A -85,B 0,C 180,E1 -696.589,E2 -696.589} C_VEL
LIN {X 0,Y 601.412,Z 135.065,A -85,B 0,C 180,E1 -699.478,E2 -699.478} C_VEL
LIN {X 0,Y 601.382,Z 135.076,A -85,B 0,C 180,E1 -702.312,E2 -702.312} C_VEL
LIN {X 0,Y 601.394,Z 135.072,A -85,B 0,C 180,E1 -704.409,E2 -704.409} C_VEL
LIN {X 0,Y 601.397,Z 135.066,A -85,B 0,C 180,E1 -707.172,E2 -707.172} C_VEL
LIN {X 0,Y 601.425,Z 135.072,A -85,B 0,C 180,E1 -709.905,E2 -709.905} C_VEL
LIN {X 0,Y 601.374,Z 135.07,A -85,B 0,C 180,E1 -712.614,E2 -712.614} C_VEL
LIN {X 0,Y 601.407,Z 135.067,A -85,B 0,C 180,E1 -715.308,E2 -715.308} C_VEL
LIN {X 0,Y 601.413,Z 135.072,A -85,B 0,C 180,E1 -717.991,E2 -717.991} C_VEL
LIN {X 0,Y 601.433,Z 135.069,A -85,B 0,C 180,E1 -720,E2 -720} C_VEL
LIN {X 0,Y 601.399,Z 135.066,A -85,B 0,C 180,E1 -722.68,E2 -722.68} C_VEL
LIN {X 0,Y 601.418,Z 135.069,A -85,B 0,C 180,E1 -725.364,E2 -725.364} C_VEL
LIN {X 0,Y 601.398,Z 135.07,A -85,B 0,C 180,E1 -728.062,E2 -728.062} C_VEL
LIN {X 0,Y 601.38,Z 135.069,A -85,B 0,C 180,E1 -730.777,E2 -730.777} C_VEL
LIN {X 0,Y 601.403,Z 135.076,A -85,B 0,C 180,E1 -733.516,E2 -733.516} C_VEL
LIN {X 0,Y 601.385,Z 135.068,A -85,B 0,C 180,E1 -736.289,E2 -736.289} C_VEL
LIN {X 0,Y 601.405,Z 135.071,A -85,B 0,C 180,E1 -739.1,E2 -739.1} C_VEL
LIN {X 0,Y 601.377,Z 135.07,A -85,B 0,C 180,E1 -741.961,E2 -741.961} C_VEL
LIN {X 0,Y 601.382,Z 135.073,A -85,B 0,C 180,E1 -744.88,E2 -744.88} C_VEL
LIN {X 0,Y 601.398,Z 135.074,A -85,B 0,C 180,E1 -747.359,E2 -747.359} C_VEL
LIN {X 0,Y 601.37,Z 135.07,A -85,B 0,C 180,E1 -750.168,E2 -750.168} C_VEL
LIN {X 0,Y 601.391,Z 135.072,A -85,B 0,C 180,E1 -752.711,E2 -752.711} C_VEL
LIN {X 0,Y 601.38,Z 135.078,A -85,B 0,C 180,E1 -755.11,E2 -755.11} C_VEL
LIN {X 0,Y 601.391,Z 135.07,A -85,B 0,C 180,E1 -757.423,E2 -757.423} C_VEL
LIN {X 0,Y 601.372,Z 135.07,A -85,B 0,C 180,E1 -759.999,E2 -759.999} C_VEL
LIN {X 0,Y 601.368,Z 135.077,A -85,B 0,C 180,E1 -762.674,E2 -762.674} C_VEL
LIN {X 0,Y 601.366,Z 135.071,A -85,B 0,C 180,E1 -765.476,E2 -765.476} C_VEL
LIN {X 0,Y 601.392,Z 135.07,A -85,B 0,C 180,E1 -768.232,E2 -768.232} C_VEL
LIN {X 0,Y 601.38,Z 135.076,A -85,B 0,C 180,E1 -770.871,E2 -770.871} C_VEL
LIN {X 0,Y 601.361,Z 135.071,A -85,B 0,C 180,E1 -773.414,E2 -773.414} C_VEL
LIN {X 0,Y 601.361,Z 135.074,A -85,B 0,C 180,E1 -776.075,E2 -776.075} C_VEL
LIN {X 0,Y 601.389,Z 135.078,A -85,B 0,C 180,E1 -778.551,E2 -778.551} C_VEL
LIN {X 0,Y 601.351,Z 135.073,A -85,B 0,C 180,E1 -781.369,E2 -781.369} C_VEL
LIN {X 0,Y 601.4,Z 135.072,A -85,B 0,C 180,E1 -784.136,E2 -784.136} C_VEL
LIN {X 0,Y 601.368,Z 135.078,A -85,B 0,C 180,E1 -786.587,E2 -786.587} C_VEL
LIN {X 0,Y 601.446,Z 135.249,A -85,B 0,C 180,E1 -788.132,E2 -788.132} C_VEL
LIN {X 0,Y 601.606,Z 141.056,A -85,B 0,C 180,E1 -789.019,E2 -789.019} C_VEL
LIN {X 0,Y 601.533,Z 158.773,A -85,B 0,C 180,E1 -791.611,E2 -791.611} C_VEL
LIN {X 0,Y 601.495,Z 176.977,A -85,B 0,C 180,E1 -794.237,E2 -794.237} C_VEL
LIN {X 0,Y 601.464,Z 195.24,A -85,B 0,C 180,E1 -796.807,E2 -796.807} C_VEL
LIN {X 0,Y 601.673,Z 198.677,A -85,B 0,C 180,E1 -796.876,E2 -796.876} C_VEL
LIN {X 0,Y 601.62,Z 302.918,A -85,B 0,C 180,E1 -798.139,E2 -798.139} C_VEL
LIN {X 0,Y 601.591,Z 316.198,A -85,B 0,C 180,E1 -798.438,E2 -798.438} C_VEL
LIN {X 0,Y 601.55,Z 327.915,A -85,B 0,C 180,E1 -798.826,E2 -798.826} C_VEL
LIN {X 0,Y 601.53,Z 338.913,A -85,B 0,C 180,E1 -799.311,E2 -799.311} C_VEL
LIN {X 0,Y 601.482,Z 349.572,A -85,B 0,C 180,E1 -799.905,E2 -799.905} C_VEL
LIN {X 0,Y 601.449,Z 360.469,A -85,B 0,C 180,E1 -800.669,E2 -800.669} C_VEL
LIN {X 0,Y 601.429,Z 371.106,A -85,B 0,C 180,E1 -801.6,E2 -801.6} C_VEL
LIN {X 0,Y 601.418,Z 378.955,A -85,B 0,C 180,E1 -802.445,E2 -802.445} C_VEL
LIN {X 0,Y 601.371,Z 386.222,A -85,B 0,C 180,E1 -803.398,E2 -803.398} C_VEL
LIN {X 0,Y 601.372,Z 391.863,A -85,B 0,C 180,E1 -804.298,E2 -804.298} C_VEL
LIN {X 0,Y 601.336,Z 396.947,A -85,B 0,C 180,E1 -805.307,E2 -805.307} C_VEL
LIN {X 0,Y 601.368,Z 400.894,A -85,B 0,C 180,E1 -806.314,E2 -806.314} C_VEL
LIN {X 0,Y 601.325,Z 403.807,A -85,B 0,C 180,E1 -807.32,E2 -807.32} C_VEL
LIN {X 0,Y 601.343,Z 405.201,A -85,B 0,C 180,E1 -807.99,E2 -807.99} C_VEL
LIN {X 0,Y 601.339,Z 406.783,A -85,B 0,C 180,E1 -809.33,E2 -809.33} C_VEL
LIN {X 0,Y 601.335,Z 407,A -85,B 0,C 180,E1 -809.999,E2 -809.999} C_VEL
LIN {X 0,Y 601.347,Z 406.185,A -85,B 0,C 180,E1 -811.339,E2 -811.339} C_VEL
LIN {X 0,Y 601.343,Z 405.203,A -85,B 0,C 180,E1 -812.009,E2 -812.009} C_VEL
LIN {X 0,Y 601.325,Z 403.811,A -85,B 0,C 180,E1 -812.679,E2 -812.679} C_VEL
LIN {X 0,Y 601.368,Z 400.899,A -85,B 0,C 180,E1 -813.685,E2 -813.685} C_VEL
LIN {X 0,Y 601.336,Z 396.953,A -85,B 0,C 180,E1 -814.692,E2 -814.692} C_VEL
LIN {X 0,Y 601.373,Z 390.882,A -85,B 0,C 180,E1 -815.868,E2 -815.868} C_VEL
LIN {X 0,Y 601.381,Z 384.242,A -85,B 0,C 180,E1 -816.879,E2 -816.879} C_VEL
LIN {X 0,Y 601.4,Z 375.997,A -85,B 0,C 180,E1 -817.891,E2 -817.891} C_VEL
LIN {X 0,Y 601.436,Z 367.546,A -85,B 0,C 180,E1 -818.737,E2 -818.737} C_VEL
LIN {X 0,Y 601.45,Z 357.105,A -85,B 0,C 180,E1 -819.584,E2 -819.584} C_VEL
LIN {X 0,Y 601.476,Z 346.773,A -85,B 0,C 180,E1 -820.263,E2 -820.263} C_VEL
LIN {X 0,Y 601.538,Z 335.908,A -85,B 0,C 180,E1 -820.835,E2 -820.835} C_VEL
LIN {X 0,Y 601.565,Z 323.397,A -85,B 0,C 180,E1 -821.34,E2 -821.34} C_VEL
LIN {X 0,Y 601.606,Z 310.39,A -85,B 0,C 180,E1 -821.71,E2 -821.71} C_VEL
LIN {X 0,Y 601.621,Z 297.152,A -85,B 0,C 180,E1 -821.945,E2 -821.945} C_VEL
LIN {X 0,Y 601.577,Z 196.26,A -85,B 0,C 180,E1 -823.157,E2 -823.157} C_VEL
LIN {X 0,Y 601.456,Z 194.978,A -85,B 0,C 180,E1 -823.213,E2 -823.213} C_VEL
LIN {X 0,Y 601.494,Z 174.56,A -85,B 0,C 180,E1 -826.11,E2 -826.11} C_VEL
LIN {X 0,Y 601.52,Z 157.176,A -85,B 0,C 180,E1 -828.621,E2 -828.621} C_VEL
LIN {X 0,Y 601.628,Z 139.365,A -85,B 0,C 180,E1 -831.23,E2 -831.23} C_VEL
LIN {X 0,Y 601.437,Z 135.186,A -85,B 0,C 180,E1 -831.889,E2 -831.889} C_VEL
LIN {X 0,Y 601.369,Z 135.071,A -85,B 0,C 180,E1 -834.879,E2 -834.879} C_VEL
LIN {X 0,Y 601.386,Z 135.074,A -85,B 0,C 180,E1 -837.356,E2 -837.356} C_VEL
LIN {X 0,Y 601.369,Z 135.072,A -85,B 0,C 180,E1 -840.166,E2 -840.166} C_VEL
LIN {X 0,Y 601.377,Z 135.069,A -85,B 0,C 180,E1 -842.708,E2 -842.708} C_VEL
LIN {X 0,Y 601.361,Z 135.075,A -85,B 0,C 180,E1 -845.107,E2 -845.107} C_VEL
LIN {X 0,Y 601.391,Z 135.078,A -85,B 0,C 180,E1 -847.421,E2 -847.421} C_VEL
LIN {X 0,Y 601.367,Z 135.072,A -85,B 0,C 180,E1 -849.997,E2 -849.997} C_VEL
LIN {X 0,Y 601.348,Z 135.073,A -85,B 0,C 180,E1 -852.584,E2 -852.584} C_VEL
LIN {X 0,Y 601.357,Z 135.072,A -85,B 0,C 180,E1 -854.528,E2 -854.528} C_VEL
LIN {X 0,Y 601.367,Z 135.078,A -85,B 0,C 180,E1 -857.412,E2 -857.412} C_VEL
LIN {X 0,Y 601.362,Z 135.071,A -85,B 0,C 180,E1 -860.001,E2 -860.001} C_VEL
LIN {X 0,Y 601.386,Z 135.07,A -85,B 0,C 180,E1 -862.622,E2 -862.622} C_VEL
LIN {X 0,Y 601.404,Z 135.075,A -85,B 0,C 180,E1 -865.067,E2 -865.067} C_VEL
LIN {X 0,Y 601.394,Z 135.071,A -85,B 0,C 180,E1 -867.482,E2 -867.482} C_VEL
LIN {X 0,Y 601.358,Z 135.072,A -85,B 0,C 180,E1 -869.86,E2 -869.86} C_VEL
LIN {X 0,Y 601.349,Z 135.072,A -85,B 0,C 180,E1 -872.129,E2 -872.129} C_VEL
LIN {X 0,Y 601.373,Z 135.071,A -85,B 0,C 180,E1 -874.379,E2 -874.379} C_VEL
LIN {X 0,Y 601.387,Z 135.072,A -85,B 0,C 180,E1 -877.316,E2 -877.316} C_VEL
LIN {X 0,Y 601.369,Z 135.071,A -85,B 0,C 180,E1 -880.189,E2 -880.189} C_VEL
LIN {X 0,Y 601.391,Z 135.075,A -85,B 0,C 180,E1 -883.013,E2 -883.013} C_VEL
LIN {X 0,Y 601.362,Z 135.071,A -85,B 0,C 180,E1 -885.793,E2 -885.793} C_VEL
LIN {X 0,Y 601.416,Z 135.071,A -85,B 0,C 180,E1 -888.541,E2 -888.541} C_VEL
LIN {X 0,Y 601.374,Z 135.071,A -85,B 0,C 180,E1 -891.261,E2 -891.261} C_VEL
LIN {X 0,Y 601.367,Z 135.071,A -85,B 0,C 180,E1 -893.384,E2 -893.384} C_VEL
LIN {X 0,Y 601.369,Z 135.071,A -85,B 0,C 180,E1 -895.307,E2 -895.307} C_VEL
LIN {X 0,Y 601.388,Z 135.068,A -85,B 0,C 180,E1 -897.32,E2 -897.32} C_VEL
LIN {X 0,Y 601.401,Z 135.068,A -85,B 0,C 180,E1 -900,E2 -900} C_VEL
LIN {X 0,Y 601.431,Z 135.07,A -85,B 0,C 180,E1 -902.679,E2 -902.679} C_VEL
LIN {X 0,Y 601.37,Z 135.07,A -85,B 0,C 180,E1 -905.364,E2 -905.364} C_VEL
LIN {X 0,Y 601.351,Z 135.072,A -85,B 0,C 180,E1 -907.386,E2 -907.386} C_VEL
LIN {X 0,Y 601.399,Z 135.071,A -85,B 0,C 180,E1 -910.095,E2 -910.095} C_VEL
LIN {X 0,Y 601.376,Z 135.073,A -85,B 0,C 180,E1 -912.381,E2 -912.381} C_VEL
LIN {X 0,Y 600.708,Z 135.155,A -85,B 0,C 180,E1 -912.94,E2 -912.94} C_VEL
LIN {X 0,Y 597.851,Z 135.511,A -85,B 0,C 180,E1 -913.848,E2 -913.848} C_VEL
LIN {X 0,Y 595.437,Z 135.815,A -85,B 0,C 180,E1 -914.578,E2 -914.578} C_VEL
LIN {X 0,Y 594.4,Z 135.939,A -85,B 0,C 180,E1 -915.142,E2 -915.142} C_VEL
LIN {X 0,Y 594.315,Z 135.949,A -85,B 0,C 180,E1 -915.333,E2 -915.333} C_VEL
LIN {X 0,Y 594.321,Z 135.948,A -85,B 0,C 180,E1 -917.195,E2 -917.195} C_VEL
LIN {X 0,Y 594.345,Z 135.952,A -85,B 0,C 180,E1 -920.054,E2 -920.054} C_VEL
LIN {X 0,Y 594.333,Z 135.947,A -85,B 0,C 180,E1 -922.968,E2 -922.968} C_VEL
LIN {X 0,Y 594.31,Z 135.949,A -85,B 0,C 180,E1 -925.196,E2 -925.196} C_VEL
LIN {X 0,Y 594.327,Z 135.949,A -85,B 0,C 180,E1 -927.519,E2 -927.519} C_VEL
LIN {X 0,Y 594.348,Z 135.948,A -85,B 0,C 180,E1 -930.561,E2 -930.561} C_VEL
LIN {X 0,Y 594.365,Z 135.963,A -85,B 0,C 180,E1 -933.66,E2 -933.66} C_VEL
LIN {X 0,Y 594.427,Z 136.326,A -85,B 0,C 180,E1 -933.829,E2 -933.829} C_VEL
LIN {X 0,Y 594.566,Z 144.31,A -85,B 0,C 180,E1 -935.154,E2 -935.154} C_VEL
LIN {X 0,Y 594.467,Z 161.462,A -85,B 0,C 180,E1 -937.934,E2 -937.934} C_VEL
LIN {X 0,Y 594.388,Z 178.861,A -85,B 0,C 180,E1 -940.691,E2 -940.691} C_VEL
LIN {X 0,Y 594.719,Z 181.39,A -85,B 0,C 180,E1 -940.762,E2 -940.762} C_VEL
LIN {X 0,Y 594.678,Z 286.393,A -85,B 0,C 180,E1 -942.052,E2 -942.052} C_VEL
LIN {X 0,Y 594.647,Z 299.775,A -85,B 0,C 180,E1 -942.363,E2 -942.363} C_VEL
LIN {X 0,Y 594.588,Z 311.365,A -85,B 0,C 180,E1 -942.758,E2 -942.758} C_VEL
LIN {X 0,Y 594.537,Z 323.011,A -85,B 0,C 180,E1 -943.284,E2 -943.284} C_VEL
LIN {X 0,Y 594.461,Z 334.585,A -85,B 0,C 180,E1 -943.961,E2 -943.961} C_VEL
LIN {X 0,Y 594.427,Z 344.558,A -85,B 0,C 180,E1 -944.692,E2 -944.692} C_VEL
LIN {X 0,Y 594.381,Z 353.38,A -85,B 0,C 180,E1 -945.477,E2 -945.477} C_VEL
LIN {X 0,Y 594.35,Z 362.216,A -85,B 0,C 180,E1 -946.432,E2 -946.432} C_VEL
LIN {X 0,Y 594.312,Z 369.385,A -85,B 0,C 180,E1 -947.388,E2 -947.388} C_VEL
LIN {X 0,Y 594.275,Z 376.217,A -85,B 0,C 180,E1 -948.529,E2 -948.529} C_VEL
LIN {X 0,Y 594.253,Z 380.484,A -85,B 0,C 180,E1 -949.425,E2 -949.425} C_VEL
LIN {X 0,Y 594.236,Z 383.869,A -85,B 0,C 180,E1 -950.31,E2 -950.31} C_VEL
LIN {X 0,Y 594.23,Z 386.756,A -85,B 0,C 180,E1 -951.314,E2 -951.314} C_VEL
LIN {X 0,Y 594.221,Z 388.834,A -85,B 0,C 180,E1 -952.412,E2 -952.412} C_VEL
LIN {X 0,Y 594.228,Z 389.938,A -85,B 0,C 180,E1 -953.748,E2 -953.748} C_VEL
LIN {X 0,Y 594.219,Z 389.804,A -85,B 0,C 180,E1 -954.694,E2 -954.694} C_VEL
LIN {X 0,Y 594.243,Z 388.526,A -85,B 0,C 180,E1 -955.881,E2 -955.881} C_VEL
LIN {X 0,Y 594.244,Z 385.9,A -85,B 0,C 180,E1 -957.108,E2 -957.108} C_VEL
LIN {X 0,Y 594.251,Z 383.649,A -85,B 0,C 180,E1 -957.847,E2 -957.847} C_VEL
LIN {X 0,Y 594.277,Z 378.805,A -85,B 0,C 180,E1 -959.042,E2 -959.042} C_VEL
LIN {X 0,Y 594.289,Z 372.466,A -85,B 0,C 180,E1 -960.22,E2 -960.22} C_VEL
LIN {X 0,Y 594.312,Z 365.659,A -85,B 0,C 180,E1 -961.221,E2 -961.221} C_VEL
LIN {X 0,Y 594.353,Z 356.854,A -85,B 0,C 180,E1 -962.262,E2 -962.262} C_VEL
LIN {X 0,Y 594.4,Z 346.875,A -85,B 0,C 180,E1 -963.208,E2 -963.208} C_VEL
LIN {X 0,Y 594.429,Z 336.96,A -85,B 0,C 180,E1 -963.968,E2 -963.968} C_VEL
LIN {X 0,Y 594.491,Z 326.373,A -85,B 0,C 180,E1 -964.626,E2 -964.626} C_VEL
LIN {X 0,Y 594.588,Z 313.654,A -85,B 0,C 180,E1 -965.243,E2 -965.243} C_VEL
LIN {X 0,Y 594.647,Z 301.281,A -85,B 0,C 180,E1 -965.683,E2 -965.683} C_VEL
LIN {X 0,Y 594.682,Z 288.556,A -85,B 0,C 180,E1 -965.997,E2 -965.997} C_VEL
LIN {X 0,Y 594.687,Z 267.338,A -85,B 0,C 180,E1 -966.287,E2 -966.287} C_VEL
LIN {X 0,Y 594.554,Z 180.251,A -85,B 0,C 180,E1 -967.346,E2 -967.346} C_VEL
LIN {X 0,Y 594.396,Z 178.641,A -85,B 0,C 180,E1 -967.42,E2 -967.42} C_VEL
LIN {X 0,Y 594.414,Z 160.522,A -85,B 0,C 180,E1 -970.309,E2 -970.309} C_VEL
LIN {X 0,Y 594.538,Z 145.075,A -85,B 0,C 180,E1 -972.812,E2 -972.812} C_VEL
LIN {X 0,Y 594.424,Z 136.098,A -85,B 0,C 180,E1 -974.31,E2 -974.31} C_VEL
LIN {X 0,Y 594.363,Z 135.943,A -85,B 0,C 180,E1 -977.018,E2 -977.018} C_VEL
LIN {X 0,Y 594.392,Z 135.947,A -85,B 0,C 180,E1 -979.785,E2 -979.785} C_VEL
LIN {X 0,Y 594.389,Z 135.941,A -85,B 0,C 180,E1 -982.528,E2 -982.528} C_VEL
LIN {X 0,Y 594.391,Z 135.941,A -85,B 0,C 180,E1 -985.253,E2 -985.253} C_VEL
LIN {X 0,Y 594.39,Z 135.947,A -85,B 0,C 180,E1 -987.968,E2 -987.968} C_VEL
LIN {X 0,Y 594.413,Z 135.936,A -85,B 0,C 180,E1 -990.678,E2 -990.678} C_VEL
LIN {X 0,Y 594.382,Z 135.946,A -85,B 0,C 180,E1 -993.39,E2 -993.39} C_VEL
LIN {X 0,Y 594.356,Z 135.946,A -85,B 0,C 180,E1 -996.11,E2 -996.11} C_VEL
LIN {X 0,Y 594.376,Z 135.942,A -85,B 0,C 180,E1 -998.843,E2 -998.843} C_VEL
LIN {X 0,Y 594.39,Z 135.948,A -85,B 0,C 180,E1 -1001.596,E2 -1001.596} C_VEL
LIN {X 0,Y 594.384,Z 135.94,A -85,B 0,C 180,E1 -1004.378,E2 -1004.378} C_VEL
LIN {X 0,Y 594.388,Z 135.947,A -85,B 0,C 180,E1 -1007.194,E2 -1007.194} C_VEL
LIN {X 0,Y 594.368,Z 135.943,A -85,B 0,C 180,E1 -1010.054,E2 -1010.054} C_VEL
LIN {X 0,Y 594.361,Z 135.949,A -85,B 0,C 180,E1 -1012.968,E2 -1012.968} C_VEL
LIN {X 0,Y 594.367,Z 135.953,A -85,B 0,C 180,E1 -1015.194,E2 -1015.194} C_VEL
LIN {X 0,Y 594.385,Z 135.944,A -85,B 0,C 180,E1 -1017.527,E2 -1017.527} C_VEL
LIN {X 0,Y 594.366,Z 135.943,A -85,B 0,C 180,E1 -1020.325,E2 -1020.325} C_VEL
LIN {X 0,Y 594.376,Z 135.95,A -85,B 0,C 180,E1 -1022.951,E2 -1022.951} C_VEL
LIN {X 0,Y 594.347,Z 135.948,A -85,B 0,C 180,E1 -1025.409,E2 -1025.409} C_VEL
LIN {X 0,Y 594.38,Z 135.941,A -85,B 0,C 180,E1 -1027.941,E2 -1027.941} C_VEL
LIN {X 0,Y 594.369,Z 135.952,A -85,B 0,C 180,E1 -1030.822,E2 -1030.822} C_VEL
LIN {X 0,Y 594.35,Z 135.947,A -85,B 0,C 180,E1 -1033.301,E2 -1033.301} C_VEL
LIN {X 0,Y 594.359,Z 135.945,A -85,B 0,C 180,E1 -1036.162,E2 -1036.162} C_VEL
LIN {X 0,Y 594.368,Z 135.945,A -85,B 0,C 180,E1 -1039.179,E2 -1039.179} C_VEL
LIN {X 0,Y 594.376,Z 135.943,A -85,B 0,C 180,E1 -1042.059,E2 -1042.059} C_VEL
LIN {X 0,Y 594.345,Z 135.953,A -85,B 0,C 180,E1 -1044.677,E2 -1044.677} C_VEL
LIN {X 0,Y 594.371,Z 135.943,A -85,B 0,C 180,E1 -1047.09,E2 -1047.09} C_VEL
LIN {X 0,Y 594.381,Z 135.941,A -85,B 0,C 180,E1 -1049.673,E2 -1049.673} C_VEL
LIN {X 0,Y 594.373,Z 135.949,A -85,B 0,C 180,E1 -1052.539,E2 -1052.539} C_VEL
LIN {X 0,Y 594.397,Z 135.939,A -85,B 0,C 180,E1 -1055.564,E2 -1055.564} C_VEL
LIN {X 0,Y 594.349,Z 135.951,A -85,B 0,C 180,E1 -1058.496,E2 -1058.496} C_VEL
LIN {X 0,Y 594.363,Z 135.943,A -85,B 0,C 180,E1 -1061.382,E2 -1061.382} C_VEL
LIN {X 0,Y 594.348,Z 135.953,A -85,B 0,C 180,E1 -1064.219,E2 -1064.219} C_VEL
LIN {X 0,Y 594.367,Z 135.948,A -85,B 0,C 180,E1 -1066.321,E2 -1066.321} C_VEL
LIN {X 0,Y 594.363,Z 135.943,A -85,B 0,C 180,E1 -1068.939,E2 -1068.939} C_VEL
LIN {X 0,Y 594.377,Z 135.949,A -85,B 0,C 180,E1 -1071.843,E2 -1071.843} C_VEL
LIN {X 0,Y 594.359,Z 135.944,A -85,B 0,C 180,E1 -1074.572,E2 -1074.572} C_VEL
LIN {X 0,Y 594.394,Z 135.941,A -85,B 0,C 180,E1 -1077.289,E2 -1077.289} C_VEL
LIN {X 0,Y 594.402,Z 135.944,A -85,B 0,C 180,E1 -1080,E2 -1080} C_VEL
LIN {X 0,Y 594.37,Z 135.942,A -85,B 0,C 180,E1 -1082.711,E2 -1082.711} C_VEL
LIN {X 0,Y 594.381,Z 135.947,A -85,B 0,C 180,E1 -1085.428,E2 -1085.428} C_VEL
LIN {X 0,Y 594.349,Z 135.947,A -85,B 0,C 180,E1 -1088.158,E2 -1088.158} C_VEL
LIN {X 0,Y 594.366,Z 135.945,A -85,B 0,C 180,E1 -1091.062,E2 -1091.062} C_VEL
LIN {X 0,Y 594.329,Z 135.948,A -85,B 0,C 180,E1 -1094.151,E2 -1094.151} C_VEL
LIN {X 0,Y 594.368,Z 135.949,A -85,B 0,C 180,E1 -1097.194,E2 -1097.194} C_VEL
LIN {X 0,Y 594.347,Z 135.946,A -85,B 0,C 180,E1 -1100.055,E2 -1100.055} C_VEL
LIN {X 0,Y 594.344,Z 135.95,A -85,B 0,C 180,E1 -1102.968,E2 -1102.968} C_VEL
LIN {X 0,Y 594.338,Z 135.947,A -85,B 0,C 180,E1 -1105.946,E2 -1105.946} C_VEL
LIN {X 0,Y 594.317,Z 135.948,A -85,B 0,C 180,E1 -1108.23,E2 -1108.23} C_VEL
LIN {X 0,Y 594.33,Z 135.949,A -85,B 0,C 180,E1 -1110.563,E2 -1110.563} C_VEL
LIN {X 0,Y 594.335,Z 135.955,A -85,B 0,C 180,E1 -1112.953,E2 -1112.953} C_VEL
LIN {X 0,Y 594.314,Z 135.953,A -85,B 0,C 180,E1 -1115.412,E2 -1115.412} C_VEL
LIN {X 0,Y 594.349,Z 135.944,A -85,B 0,C 180,E1 -1117.944,E2 -1117.944} C_VEL
LIN {X 0,Y 594.345,Z 135.954,A -85,B 0,C 180,E1 -1120.818,E2 -1120.818} C_VEL
LIN {X 0,Y 594.332,Z 135.947,A -85,B 0,C 180,E1 -1123.836,E2 -1123.836} C_VEL
LIN {X 0,Y 594.34,Z 135.955,A -85,B 0,C 180,E1 -1126.698,E2 -1126.698} C_VEL
LIN {X 0,Y 594.315,Z 135.949,A -85,B 0,C 180,E1 -1129.428,E2 -1129.428} C_VEL
LIN {X 0,Y 594.348,Z 135.951,A -85,B 0,C 180,E1 -1132.397,E2 -1132.397} C_VEL
LIN {X 0,Y 594.296,Z 135.951,A -85,B 0,C 180,E1 -1135.414,E2 -1135.414} C_VEL
LIN {X 0,Y 594.329,Z 135.948,A -85,B 0,C 180,E1 -1137.85,E2 -1137.85} C_VEL
LIN {X 0,Y 594.336,Z 135.952,A -85,B 0,C 180,E1 -1140.221,E2 -1140.221} C_VEL
LIN {X 0,Y 594.338,Z 135.946,A -85,B 0,C 180,E1 -1143.298,E2 -1143.298} C_VEL
LIN {X 0,Y 594.34,Z 135.956,A -85,B 0,C 180,E1 -1146.293,E2 -1146.293} C_VEL
LIN {X 0,Y 594.389,Z 136.147,A -85,B 0,C 180,E1 -1147.996,E2 -1147.996} C_VEL
LIN {X 0,Y 594.691,Z 140.485,A -85,B 0,C 180,E1 -1148.678,E2 -1148.678} C_VEL
LIN {X 0,Y 594.542,Z 158.773,A -85,B 0,C 180,E1 -1151.387,E2 -1151.387} C_VEL
LIN {X 0,Y 594.503,Z 175.764,A -85,B 0,C 180,E1 -1153.87,E2 -1153.87} C_VEL
LIN {X 0,Y 594.434,Z 195.232,A -85,B 0,C 180,E1 -1156.648,E2 -1156.648} C_VEL
LIN {X 0,Y 594.772,Z 198.677,A -85,B 0,C 180,E1 -1156.721,E2 -1156.721} C_VEL
LIN {X 0,Y 594.673,Z 302.918,A -85,B 0,C 180,E1 -1157.999,E2 -1157.999} C_VEL
LIN {X 0,Y 594.64,Z 316.199,A -85,B 0,C 180,E1 -1158.301,E2 -1158.301} C_VEL
LIN {X 0,Y 594.588,Z 329.362,A -85,B 0,C 180,E1 -1158.749,E2 -1158.749} C_VEL
LIN {X 0,Y 594.537,Z 340.621,A -85,B 0,C 180,E1 -1159.27,E2 -1159.27} C_VEL
LIN {X 0,Y 594.483,Z 352.193,A -85,B 0,C 180,E1 -1159.957,E2 -1159.957} C_VEL
LIN {X 0,Y 594.414,Z 362.59,A -85,B 0,C 180,E1 -1160.729,E2 -1160.729} C_VEL
LIN {X 0,Y 594.366,Z 371.106,A -85,B 0,C 180,E1 -1161.5,E2 -1161.5} C_VEL
LIN {X 0,Y 594.347,Z 378.955,A -85,B 0,C 180,E1 -1162.355,E2 -1162.355} C_VEL
LIN {X 0,Y 594.283,Z 386.811,A -85,B 0,C 180,E1 -1163.408,E2 -1163.408} C_VEL
LIN {X 0,Y 594.289,Z 393.677,A -85,B 0,C 180,E1 -1164.571,E2 -1164.571} C_VEL
LIN {X 0,Y 594.27,Z 398.369,A -85,B 0,C 180,E1 -1165.591,E2 -1165.591} C_VEL
LIN {X 0,Y 594.267,Z 401.954,A -85,B 0,C 180,E1 -1166.609,E2 -1166.609} C_VEL
LIN {X 0,Y 594.226,Z 403.807,A -85,B 0,C 180,E1 -1167.288,E2 -1167.288} C_VEL
LIN {X 0,Y 594.242,Z 405.199,A -85,B 0,C 180,E1 -1167.966,E2 -1167.966} C_VEL
LIN {X 0,Y 594.239,Z 406.784,A -85,B 0,C 180,E1 -1169.322,E2 -1169.322} C_VEL
LIN {X 0,Y 594.236,Z 407,A -85,B 0,C 180,E1 -1169.999,E2 -1169.999} C_VEL
LIN {X 0,Y 594.247,Z 406.186,A -85,B 0,C 180,E1 -1171.355,E2 -1171.355} C_VEL
LIN {X 0,Y 594.242,Z 405.202,A -85,B 0,C 180,E1 -1172.033,E2 -1172.033} C_VEL
LIN {X 0,Y 594.226,Z 403.811,A -85,B 0,C 180,E1 -1172.711,E2 -1172.711} C_VEL
LIN {X 0,Y 594.289,Z 400.898,A -85,B 0,C 180,E1 -1173.729,E2 -1173.729} C_VEL
LIN {X 0,Y 594.241,Z 396.953,A -85,B 0,C 180,E1 -1174.748,E2 -1174.748} C_VEL
LIN {X 0,Y 594.305,Z 390.882,A -85,B 0,C 180,E1 -1175.938,E2 -1175.938} C_VEL
LIN {X 0,Y 594.307,Z 384.242,A -85,B 0,C 180,E1 -1176.961,E2 -1176.961} C_VEL
LIN {X 0,Y 594.359,Z 375.997,A -85,B 0,C 180,E1 -1177.986,E2 -1177.986} C_VEL
LIN {X 0,Y 594.382,Z 367.547,A -85,B 0,C 180,E1 -1178.841,E2 -1178.841} C_VEL
LIN {X 0,Y 594.434,Z 357.107,A -85,B 0,C 180,E1 -1179.698,E2 -1179.698} C_VEL
LIN {X 0,Y 594.491,Z 346.773,A -85,B 0,C 180,E1 -1180.385,E2 -1180.385} C_VEL
LIN {X 0,Y 594.562,Z 335.685,A -85,B 0,C 180,E1 -1180.975,E2 -1180.975} C_VEL
LIN {X 0,Y 594.599,Z 323.721,A -85,B 0,C 180,E1 -1181.463,E2 -1181.463} C_VEL
LIN {X 0,Y 594.653,Z 310.389,A -85,B 0,C 180,E1 -1181.849,E2 -1181.849} C_VEL
LIN {X 0,Y 594.695,Z 297.152,A -85,B 0,C 180,E1 -1182.086,E2 -1182.086} C_VEL
LIN {X 0,Y 594.659,Z 197.008,A -85,B 0,C 180,E1 -1183.302,E2 -1183.302} C_VEL
LIN {X 0,Y 594.427,Z 194.975,A -85,B 0,C 180,E1 -1183.372,E2 -1183.372} C_VEL
LIN {X 0,Y 594.502,Z 175.774,A -85,B 0,C 180,E1 -1186.128,E2 -1186.128} C_VEL
LIN {X 0,Y 594.585,Z 157.012,A -85,B 0,C 180,E1 -1188.871,E2 -1188.871} C_VEL
LIN {X 0,Y 594.695,Z 139.365,A -85,B 0,C 180,E1 -1191.49,E2 -1191.49} C_VEL
LIN {X 0,Y 594.38,Z 136.076,A -85,B 0,C 180,E1 -1192.026,E2 -1192.026} C_VEL
LIN {X 0,Y 594.338,Z 135.947,A -85,B 0,C 180,E1 -1194.447,E2 -1194.447} C_VEL
LIN {X 0,Y 594.344,Z 135.946,A -85,B 0,C 180,E1 -1196.7,E2 -1196.7} C_VEL
LIN {X 0,Y 594.334,Z 135.953,A -85,B 0,C 180,E1 -1199.777,E2 -1199.777} C_VEL
LIN {X 0,Y 594.329,Z 135.949,A -85,B 0,C 180,E1 -1202.148,E2 -1202.148} C_VEL
LIN {X 0,Y 594.345,Z 135.945,A -85,B 0,C 180,E1 -1204.581,E2 -1204.581} C_VEL
LIN {X 0,Y 594.348,Z 135.952,A -85,B 0,C 180,E1 -1207.603,E2 -1207.603} C_VEL
LIN {X 0,Y 594.331,Z 135.947,A -85,B 0,C 180,E1 -1210.568,E2 -1210.568} C_VEL
LIN {X 0,Y 594.333,Z 135.956,A -85,B 0,C 180,E1 -1213.301,E2 -1213.301} C_VEL
LIN {X 0,Y 594.33,Z 135.947,A -85,B 0,C 180,E1 -1216.162,E2 -1216.162} C_VEL
LIN {X 0,Y 594.352,Z 135.954,A -85,B 0,C 180,E1 -1219.179,E2 -1219.179} C_VEL
LIN {X 0,Y 594.343,Z 135.945,A -85,B 0,C 180,E1 -1222.056,E2 -1222.056} C_VEL
LIN {X 0,Y 594.319,Z 135.951,A -85,B 0,C 180,E1 -1224.678,E2 -1224.678} C_VEL
LIN {X 0,Y 594.329,Z 135.957,A -85,B 0,C 180,E1 -1227.093,E2 -1227.093} C_VEL
LIN {X 0,Y 594.335,Z 135.948,A -85,B 0,C 180,E1 -1229.678,E2 -1229.678} C_VEL
LIN {X 0,Y 594.313,Z 135.949,A -85,B 0,C 180,E1 -1231.769,E2 -1231.769} C_VEL
LIN {X 0,Y 594.325,Z 135.947,A -85,B 0,C 180,E1 -1234.053,E2 -1234.053} C_VEL
LIN {X 0,Y 594.332,Z 135.956,A -85,B 0,C 180,E1 -1237.031,E2 -1237.031} C_VEL
LIN {X 0,Y 594.337,Z 135.946,A -85,B 0,C 180,E1 -1239.945,E2 -1239.945} C_VEL
LIN {X 0,Y 594.356,Z 135.953,A -85,B 0,C 180,E1 -1242.805,E2 -1242.805} C_VEL
LIN {X 0,Y 594.326,Z 135.947,A -85,B 0,C 180,E1 -1245.621,E2 -1245.621} C_VEL
LIN {X 0,Y 594.371,Z 135.946,A -85,B 0,C 180,E1 -1248.404,E2 -1248.404} C_VEL
LIN {X 0,Y 594.347,Z 135.948,A -85,B 0,C 180,E1 -1251.157,E2 -1251.157} C_VEL
LIN {X 0,Y 594.342,Z 135.946,A -85,B 0,C 180,E1 -1253.343,E2 -1253.343} C_VEL
LIN {X 0,Y 594.344,Z 135.947,A -85,B 0,C 180,E1 -1255.252,E2 -1255.252} C_VEL
LIN {X 0,Y 594.352,Z 135.945,A -85,B 0,C 180,E1 -1257.967,E2 -1257.967} C_VEL
LIN {X 0,Y 594.408,Z 135.945,A -85,B 0,C 180,E1 -1260.677,E2 -1260.677} C_VEL
LIN {X 0,Y 594.298,Z 135.951,A -85,B 0,C 180,E1 -1263.389,E2 -1263.389} C_VEL
LIN {X 0,Y 594.339,Z 135.946,A -85,B 0,C 180,E1 -1265.428,E2 -1265.428} C_VEL
LIN {X 0,Y 594.324,Z 135.948,A -85,B 0,C 180,E1 -1267.474,E2 -1267.474} C_VEL
LIN {X 0,Y 594.358,Z 135.951,A -85,B 0,C 180,E1 -1270.216,E2 -1270.216} C_VEL
LIN {X 0,Y 594.329,Z 135.948,A -85,B 0,C 180,E1 -1272.984,E2 -1272.984} C_VEL
LIN {X 0,Y 594.315,Z 135.949,A -85,B 0,C 180,E1 -1275.333,E2 -1275.333} C_VEL
LIN {X 0,Y 593.644,Z 136.037,A -85,B 0,C 180,E1 -1275.898,E2 -1275.898} C_VEL
LIN {X 0,Y 590.776,Z 136.398,A -85,B 0,C 180,E1 -1276.816,E2 -1276.816} C_VEL
LIN {X 0,Y 588.365,Z 136.7,A -85,B 0,C 180,E1 -1277.554,E2 -1277.554} C_VEL
LIN {X 0,Y 587.344,Z 136.825,A -85,B 0,C 180,E1 -1278.124,E2 -1278.124} C_VEL
LIN {X 0,Y 587.269,Z 136.832,A -85,B 0,C 180,E1 -1278.317,E2 -1278.317} C_VEL
LIN {X 0,Y 587.316,Z 136.821,A -85,B 0,C 180,E1 -1281.038,E2 -1281.038} C_VEL
LIN {X 0,Y 587.311,Z 136.829,A -85,B 0,C 180,E1 -1284.007,E2 -1284.007} C_VEL
LIN {X 0,Y 587.287,Z 136.832,A -85,B 0,C 180,E1 -1286.281,E2 -1286.281} C_VEL
LIN {X 0,Y 587.284,Z 136.825,A -85,B 0,C 180,E1 -1289.125,E2 -1289.125} C_VEL
LIN {X 0,Y 587.299,Z 136.831,A -85,B 0,C 180,E1 -1291.831,E2 -1291.831} C_VEL
LIN {X 0,Y 587.347,Z 136.999,A -85,B 0,C 180,E1 -1293.678,E2 -1293.678} C_VEL
LIN {X 0,Y 587.609,Z 139.986,A -85,B 0,C 180,E1 -1294.203,E2 -1294.203} C_VEL
LIN {X 0,Y 587.477,Z 157.967,A -85,B 0,C 180,E1 -1297.166,E2 -1297.166} C_VEL
LIN {X 0,Y 587.373,Z 174.532,A -85,B 0,C 180,E1 -1299.856,E2 -1299.856} C_VEL
LIN {X 0,Y 587.404,Z 179.046,A -85,B 0,C 180,E1 -1300.542,E2 -1300.542} C_VEL
LIN {X 0,Y 587.855,Z 183.616,A -85,B 0,C 180,E1 -1300.631,E2 -1300.631} C_VEL
LIN {X 0,Y 587.738,Z 286.577,A -85,B 0,C 180,E1 -1301.911,E2 -1301.911} C_VEL
LIN {X 0,Y 587.7,Z 299.795,A -85,B 0,C 180,E1 -1302.225,E2 -1302.225} C_VEL
LIN {X 0,Y 587.632,Z 310.359,A -85,B 0,C 180,E1 -1302.584,E2 -1302.584} C_VEL
LIN {X 0,Y 587.555,Z 321.444,A -85,B 0,C 180,E1 -1303.076,E2 -1303.076} C_VEL
LIN {X 0,Y 587.474,Z 333.819,A -85,B 0,C 180,E1 -1303.788,E2 -1303.788} C_VEL
LIN {X 0,Y 587.382,Z 345.021,A -85,B 0,C 180,E1 -1304.618,E2 -1304.618} C_VEL
LIN {X 0,Y 587.329,Z 353.776,A -85,B 0,C 180,E1 -1305.414,E2 -1305.414} C_VEL
LIN {X 0,Y 587.274,Z 361.616,A -85,B 0,C 180,E1 -1306.271,E2 -1306.271} C_VEL
LIN {X 0,Y 587.24,Z 368.82,A -85,B 0,C 180,E1 -1307.223,E2 -1307.223} C_VEL
LIN {X 0,Y 587.207,Z 375.768,A -85,B 0,C 180,E1 -1308.377,E2 -1308.377} C_VEL
LIN {X 0,Y 587.167,Z 380.356,A -85,B 0,C 180,E1 -1309.339,E2 -1309.339} C_VEL
LIN {X 0,Y 587.137,Z 384.002,A -85,B 0,C 180,E1 -1310.31,E2 -1310.31} C_VEL
LIN {X 0,Y 587.118,Z 387.232,A -85,B 0,C 180,E1 -1311.506,E2 -1311.506} C_VEL
LIN {X 0,Y 587.135,Z 388.807,A -85,B 0,C 180,E1 -1312.378,E2 -1312.378} C_VEL
LIN {X 0,Y 587.118,Z 389.762,A -85,B 0,C 180,E1 -1313.322,E2 -1313.322} C_VEL
LIN {X 0,Y 587.128,Z 389.889,A -85,B 0,C 180,E1 -1314.485,E2 -1314.485} C_VEL
LIN {X 0,Y 587.14,Z 388.736,A -85,B 0,C 180,E1 -1315.767,E2 -1315.767} C_VEL
LIN {X 0,Y 587.137,Z 386.488,A -85,B 0,C 180,E1 -1316.918,E2 -1316.918} C_VEL
LIN {X 0,Y 587.179,Z 382.472,A -85,B 0,C 180,E1 -1318.223,E2 -1318.223} C_VEL
LIN {X 0,Y 587.211,Z 377.866,A -85,B 0,C 180,E1 -1319.299,E2 -1319.299} C_VEL
LIN {X 0,Y 587.229,Z 371.706,A -85,B 0,C 180,E1 -1320.418,E2 -1320.418} C_VEL
LIN {X 0,Y 587.239,Z 364.98,A -85,B 0,C 180,E1 -1321.4,E2 -1321.4} C_VEL
LIN {X 0,Y 587.325,Z 356.079,A -85,B 0,C 180,E1 -1322.445,E2 -1322.445} C_VEL
LIN {X 0,Y 587.37,Z 346.586,A -85,B 0,C 180,E1 -1323.341,E2 -1323.341} C_VEL
LIN {X 0,Y 587.404,Z 336.666,A -85,B 0,C 180,E1 -1324.107,E2 -1324.107} C_VEL
LIN {X 0,Y 587.507,Z 325.952,A -85,B 0,C 180,E1 -1324.777,E2 -1324.777} C_VEL
LIN {X 0,Y 587.612,Z 313.093,A -85,B 0,C 180,E1 -1325.4,E2 -1325.4} C_VEL
LIN {X 0,Y 587.666,Z 300.898,A -85,B 0,C 180,E1 -1325.833,E2 -1325.833} C_VEL
LIN {X 0,Y 587.756,Z 288.491,A -85,B 0,C 180,E1 -1326.142,E2 -1326.142} C_VEL
LIN {X 0,Y 587.759,Z 267.256,A -85,B 0,C 180,E1 -1326.434,E2 -1326.434} C_VEL
LIN {X 0,Y 587.718,Z 181.434,A -85,B 0,C 180,E1 -1327.489,E2 -1327.489} C_VEL
LIN {X 0,Y 587.394,Z 178.887,A -85,B 0,C 180,E1 -1327.559,E2 -1327.559} C_VEL
LIN {X 0,Y 587.425,Z 161.005,A -85,B 0,C 180,E1 -1330.429,E2 -1330.429} C_VEL
LIN {X 0,Y 587.565,Z 144.641,A -85,B 0,C 180,E1 -1333.115,E2 -1333.115} C_VEL
LIN {X 0,Y 587.609,Z 139.103,A -85,B 0,C 180,E1 -1334.034,E2 -1334.034} C_VEL
LIN {X 0,Y 587.349,Z 136.883,A -85,B 0,C 180,E1 -1334.472,E2 -1334.472} C_VEL
LIN {X 0,Y 587.314,Z 136.822,A -85,B 0,C 180,E1 -1336.859,E2 -1336.859} C_VEL
LIN {X 0,Y 587.341,Z 136.823,A -85,B 0,C 180,E1 -1339.661,E2 -1339.661} C_VEL
LIN {X 0,Y 587.363,Z 136.817,A -85,B 0,C 180,E1 -1342.438,E2 -1342.438} C_VEL
LIN {X 0,Y 587.36,Z 136.816,A -85,B 0,C 180,E1 -1345.196,E2 -1345.196} C_VEL
LIN {X 0,Y 587.361,Z 136.823,A -85,B 0,C 180,E1 -1347.944,E2 -1347.944} C_VEL
LIN {X 0,Y 587.384,Z 136.812,A -85,B 0,C 180,E1 -1350.686,E2 -1350.686} C_VEL
LIN {X 0,Y 587.333,Z 136.825,A -85,B 0,C 180,E1 -1353.431,E2 -1353.431} C_VEL
LIN {X 0,Y 587.355,Z 136.824,A -85,B 0,C 180,E1 -1355.494,E2 -1355.494} C_VEL
LIN {X 0,Y 587.338,Z 136.819,A -85,B 0,C 180,E1 -1358.256,E2 -1358.256} C_VEL
LIN {X 0,Y 587.347,Z 136.821,A -85,B 0,C 180,E1 -1361.134,E2 -1361.134} C_VEL
LIN {X 0,Y 587.355,Z 136.816,A -85,B 0,C 180,E1 -1364.257,E2 -1364.257} C_VEL
LIN {X 0,Y 587.346,Z 136.827,A -85,B 0,C 180,E1 -1367.407,E2 -1367.407} C_VEL
LIN {X 0,Y 587.325,Z 136.819,A -85,B 0,C 180,E1 -1370.305,E2 -1370.305} C_VEL
LIN {X 0,Y 587.316,Z 136.831,A -85,B 0,C 180,E1 -1373.259,E2 -1373.259} C_VEL
LIN {X 0,Y 587.324,Z 136.824,A -85,B 0,C 180,E1 -1375.517,E2 -1375.517} C_VEL
LIN {X 0,Y 587.346,Z 136.818,A -85,B 0,C 180,E1 -1377.818,E2 -1377.818} C_VEL
LIN {X 0,Y 587.321,Z 136.822,A -85,B 0,C 180,E1 -1380.508,E2 -1380.508} C_VEL
LIN {X 0,Y 587.336,Z 136.827,A -85,B 0,C 180,E1 -1383.112,E2 -1383.112} C_VEL
LIN {X 0,Y 587.288,Z 136.824,A -85,B 0,C 180,E1 -1385.901,E2 -1385.901} C_VEL
LIN {X 0,Y 587.325,Z 136.823,A -85,B 0,C 180,E1 -1388.48,E2 -1388.48} C_VEL
LIN {X 0,Y 587.33,Z 136.824,A -85,B 0,C 180,E1 -1391.158,E2 -1391.158} C_VEL
LIN {X 0,Y 587.316,Z 136.822,A -85,B 0,C 180,E1 -1394.113,E2 -1394.113} C_VEL
LIN {X 0,Y 587.296,Z 136.829,A -85,B 0,C 180,E1 -1396.992,E2 -1396.992} C_VEL
LIN {X 0,Y 587.306,Z 136.822,A -85,B 0,C 180,E1 -1399.745,E2 -1399.745} C_VEL
LIN {X 0,Y 587.339,Z 136.824,A -85,B 0,C 180,E1 -1402.392,E2 -1402.392} C_VEL
LIN {X 0,Y 587.352,Z 136.817,A -85,B 0,C 180,E1 -1405.78,E2 -1405.78} C_VEL
LIN {X 0,Y 587.333,Z 136.824,A -85,B 0,C 180,E1 -1408.231,E2 -1408.231} C_VEL
LIN {X 0,Y 587.342,Z 136.821,A -85,B 0,C 180,E1 -1410.868,E2 -1410.868} C_VEL
LIN {X 0,Y 587.309,Z 136.824,A -85,B 0,C 180,E1 -1413.829,E2 -1413.829} C_VEL
LIN {X 0,Y 587.326,Z 136.824,A -85,B 0,C 180,E1 -1415.993,E2 -1415.993} C_VEL
LIN {X 0,Y 587.33,Z 136.82,A -85,B 0,C 180,E1 -1418.963,E2 -1418.963} C_VEL
LIN {X 0,Y 587.292,Z 136.829,A -85,B 0,C 180,E1 -1421.873,E2 -1421.873} C_VEL
LIN {X 0,Y 587.302,Z 136.831,A -85,B 0,C 180,E1 -1424.025,E2 -1424.025} C_VEL
LIN {X 0,Y 587.349,Z 136.826,A -85,B 0,C 180,E1 -1426.154,E2 -1426.154} C_VEL
LIN {X 0,Y 587.336,Z 136.818,A -85,B 0,C 180,E1 -1428.963,E2 -1428.963} C_VEL
LIN {X 0,Y 587.336,Z 136.824,A -85,B 0,C 180,E1 -1431.745,E2 -1431.745} C_VEL
LIN {X 0,Y 587.328,Z 136.821,A -85,B 0,C 180,E1 -1434.507,E2 -1434.507} C_VEL
LIN {X 0,Y 587.358,Z 136.817,A -85,B 0,C 180,E1 -1437.257,E2 -1437.257} C_VEL
LIN {X 0,Y 587.371,Z 136.82,A -85,B 0,C 180,E1 -1440,E2 -1440} C_VEL
LIN {X 0,Y 587.34,Z 136.817,A -85,B 0,C 180,E1 -1442.744,E2 -1442.744} C_VEL
LIN {X 0,Y 587.345,Z 136.824,A -85,B 0,C 180,E1 -1445.493,E2 -1445.493} C_VEL
LIN {X 0,Y 587.314,Z 136.822,A -85,B 0,C 180,E1 -1448.256,E2 -1448.256} C_VEL
LIN {X 0,Y 587.33,Z 136.822,A -85,B 0,C 180,E1 -1451.125,E2 -1451.125} C_VEL
LIN {X 0,Y 587.3,Z 136.823,A -85,B 0,C 180,E1 -1454.236,E2 -1454.236} C_VEL
LIN {X 0,Y 587.319,Z 136.822,A -85,B 0,C 180,E1 -1456.805,E2 -1456.805} C_VEL
LIN {X 0,Y 587.297,Z 136.829,A -85,B 0,C 180,E1 -1459.577,E2 -1459.577} C_VEL
LIN {X 0,Y 587.301,Z 136.825,A -85,B 0,C 180,E1 -1461.775,E2 -1461.775} C_VEL
LIN {X 0,Y 587.293,Z 136.826,A -85,B 0,C 180,E1 -1464.761,E2 -1464.761} C_VEL
LIN {X 0,Y 587.296,Z 136.826,A -85,B 0,C 180,E1 -1467.683,E2 -1467.683} C_VEL
LIN {X 0,Y 587.288,Z 136.826,A -85,B 0,C 180,E1 -1470.502,E2 -1470.502} C_VEL
LIN {X 0,Y 587.282,Z 136.835,A -85,B 0,C 180,E1 -1473.103,E2 -1473.103} C_VEL
LIN {X 0,Y 587.262,Z 136.83,A -85,B 0,C 180,E1 -1475.533,E2 -1475.533} C_VEL
LIN {X 0,Y 587.306,Z 136.822,A -85,B 0,C 180,E1 -1477.834,E2 -1477.834} C_VEL
LIN {X 0,Y 587.276,Z 136.827,A -85,B 0,C 180,E1 -1480.258,E2 -1480.258} C_VEL
LIN {X 0,Y 587.284,Z 136.83,A -85,B 0,C 180,E1 -1483.115,E2 -1483.115} C_VEL
LIN {X 0,Y 587.287,Z 136.825,A -85,B 0,C 180,E1 -1486.046,E2 -1486.046} C_VEL
LIN {X 0,Y 587.29,Z 136.83,A -85,B 0,C 180,E1 -1488.931,E2 -1488.931} C_VEL
LIN {X 0,Y 587.266,Z 136.827,A -85,B 0,C 180,E1 -1491.515,E2 -1491.515} C_VEL
LIN {X 0,Y 587.252,Z 136.831,A -85,B 0,C 180,E1 -1494.097,E2 -1494.097} C_VEL
LIN {X 0,Y 587.282,Z 136.829,A -85,B 0,C 180,E1 -1496.897,E2 -1496.897} C_VEL
LIN {X 0,Y 587.285,Z 136.825,A -85,B 0,C 180,E1 -1499.499,E2 -1499.499} C_VEL
LIN {X 0,Y 587.285,Z 136.834,A -85,B 0,C 180,E1 -1502.32,E2 -1502.32} C_VEL
LIN {X 0,Y 587.307,Z 136.831,A -85,B 0,C 180,E1 -1504.482,E2 -1504.482} C_VEL
LIN {X 0,Y 587.275,Z 136.832,A -85,B 0,C 180,E1 -1507.483,E2 -1507.483} C_VEL
LIN {X 0,Y 587.334,Z 137.028,A -85,B 0,C 180,E1 -1507.856,E2 -1507.856} C_VEL
LIN {X 0,Y 587.771,Z 140.561,A -85,B 0,C 180,E1 -1508.426,E2 -1508.426} C_VEL
LIN {X 0,Y 587.602,Z 158.773,A -85,B 0,C 180,E1 -1511.159,E2 -1511.159} C_VEL
LIN {X 0,Y 587.503,Z 175.764,A -85,B 0,C 180,E1 -1513.673,E2 -1513.673} C_VEL
LIN {X 0,Y 587.412,Z 195.231,A -85,B 0,C 180,E1 -1516.486,E2 -1516.486} C_VEL
LIN {X 0,Y 587.871,Z 198.677,A -85,B 0,C 180,E1 -1516.563,E2 -1516.563} C_VEL
LIN {X 0,Y 587.734,Z 302.918,A -85,B 0,C 180,E1 -1517.855,E2 -1517.855} C_VEL
LIN {X 0,Y 587.685,Z 316.2,A -85,B 0,C 180,E1 -1518.16,E2 -1518.16} C_VEL
LIN {X 0,Y 587.603,Z 328.762,A -85,B 0,C 180,E1 -1518.59,E2 -1518.59} C_VEL
LIN {X 0,Y 587.54,Z 340.619,A -85,B 0,C 180,E1 -1519.14,E2 -1519.14} C_VEL
LIN {X 0,Y 587.471,Z 352.195,A -85,B 0,C 180,E1 -1519.836,E2 -1519.836} C_VEL
LIN {X 0,Y 587.366,Z 362.592,A -85,B 0,C 180,E1 -1520.617,E2 -1520.617} C_VEL
LIN {X 0,Y 587.31,Z 371.106,A -85,B 0,C 180,E1 -1521.397,E2 -1521.397} C_VEL
LIN {X 0,Y 587.274,Z 378.955,A -85,B 0,C 180,E1 -1522.262,E2 -1522.262} C_VEL
LIN {X 0,Y 587.231,Z 385.464,A -85,B 0,C 180,E1 -1523.126,E2 -1523.126} C_VEL
LIN {X 0,Y 587.237,Z 391.863,A -85,B 0,C 180,E1 -1524.161,E2 -1524.161} C_VEL
LIN {X 0,Y 587.147,Z 396.947,A -85,B 0,C 180,E1 -1525.193,E2 -1525.193} C_VEL
LIN {X 0,Y 587.213,Z 400.893,A -85,B 0,C 180,E1 -1526.225,E2 -1526.225} C_VEL
LIN {X 0,Y 587.132,Z 403.807,A -85,B 0,C 180,E1 -1527.255,E2 -1527.255} C_VEL
LIN {X 0,Y 587.141,Z 405.198,A -85,B 0,C 180,E1 -1527.941,E2 -1527.941} C_VEL
LIN {X 0,Y 587.14,Z 406.784,A -85,B 0,C 180,E1 -1529.313,E2 -1529.313} C_VEL
LIN {X 0,Y 587.137,Z 407,A -85,B 0,C 180,E1 -1529.999,E2 -1529.999} C_VEL
LIN {X 0,Y 587.147,Z 406.187,A -85,B 0,C 180,E1 -1531.371,E2 -1531.371} C_VEL
LIN {X 0,Y 587.141,Z 405.202,A -85,B 0,C 180,E1 -1532.057,E2 -1532.057} C_VEL
LIN {X 0,Y 587.132,Z 403.812,A -85,B 0,C 180,E1 -1532.744,E2 -1532.744} C_VEL
LIN {X 0,Y 587.213,Z 400.898,A -85,B 0,C 180,E1 -1533.774,E2 -1533.774} C_VEL
LIN {X 0,Y 587.147,Z 396.952,A -85,B 0,C 180,E1 -1534.806,E2 -1534.806} C_VEL
LIN {X 0,Y 587.218,Z 390.882,A -85,B 0,C 180,E1 -1536.01,E2 -1536.01} C_VEL
LIN {X 0,Y 587.244,Z 384.243,A -85,B 0,C 180,E1 -1537.045,E2 -1537.045} C_VEL
LIN {X 0,Y 587.299,Z 375.998,A -85,B 0,C 180,E1 -1538.082,E2 -1538.082} C_VEL
LIN {X 0,Y 587.343,Z 367.547,A -85,B 0,C 180,E1 -1538.948,E2 -1538.948} C_VEL
LIN {X 0,Y 587.422,Z 357.108,A -85,B 0,C 180,E1 -1539.815,E2 -1539.815} C_VEL
LIN {X 0,Y 587.512,Z 346.771,A -85,B 0,C 180,E1 -1540.51,E2 -1540.51} C_VEL
LIN {X 0,Y 587.583,Z 334.816,A -85,B 0,C 180,E1 -1541.148,E2 -1541.148} C_VEL
LIN {X 0,Y 587.636,Z 322.615,A -85,B 0,C 180,E1 -1541.639,E2 -1541.639} C_VEL
LIN {X 0,Y 587.709,Z 309.473,A -85,B 0,C 180,E1 -1542.013,E2 -1542.013} C_VEL
LIN {X 0,Y 587.765,Z 297.152,A -85,B 0,C 180,E1 -1542.231,E2 -1542.231} C_VEL
LIN {X 0,Y 587.755,Z 197.679,A -85,B 0,C 180,E1 -1543.452,E2 -1543.452} C_VEL
LIN {X 0,Y 587.386,Z 195.253,A -85,B 0,C 180,E1 -1543.513,E2 -1543.513} C_VEL
LIN {X 0,Y 587.484,Z 178.201,A -85,B 0,C 180,E1 -1545.97,E2 -1545.97} C_VEL
LIN {X 0,Y 587.584,Z 161.21,A -85,B 0,C 180,E1 -1548.478,E2 -1548.478} C_VEL
LIN {X 0,Y 587.736,Z 143.44,A -85,B 0,C 180,E1 -1551.139,E2 -1551.139} C_VEL
LIN {X 0,Y 587.553,Z 138.128,A -85,B 0,C 180,E1 -1551.949,E2 -1551.949} C_VEL
LIN {X 0,Y 587.302,Z 136.907,A -85,B 0,C 180,E1 -1552.19,E2 -1552.19} C_VEL
LIN {X 0,Y 587.297,Z 136.825,A -85,B 0,C 180,E1 -1554.76,E2 -1554.76} C_VEL
LIN {X 0,Y 587.29,Z 136.834,A -85,B 0,C 180,E1 -1557.681,E2 -1557.681} C_VEL
LIN {X 0,Y 587.281,Z 136.825,A -85,B 0,C 180,E1 -1560.5,E2 -1560.5} C_VEL
LIN {X 0,Y 587.325,Z 136.824,A -85,B 0,C 180,E1 -1563.109,E2 -1563.109} C_VEL
LIN {X 0,Y 587.265,Z 136.831,A -85,B 0,C 180,E1 -1565.9,E2 -1565.9} C_VEL
LIN {X 0,Y 587.264,Z 136.827,A -85,B 0,C 180,E1 -1568.483,E2 -1568.483} C_VEL
LIN {X 0,Y 587.302,Z 136.829,A -85,B 0,C 180,E1 -1571.158,E2 -1571.158} C_VEL
LIN {X 0,Y 587.277,Z 136.826,A -85,B 0,C 180,E1 -1574.108,E2 -1574.108} C_VEL
LIN {X 0,Y 587.277,Z 136.831,A -85,B 0,C 180,E1 -1576.99,E2 -1576.99} C_VEL
LIN {X 0,Y 587.287,Z 136.827,A -85,B 0,C 180,E1 -1579.743,E2 -1579.743} C_VEL
LIN {X 0,Y 587.299,Z 136.823,A -85,B 0,C 180,E1 -1582.389,E2 -1582.389} C_VEL
LIN {X 0,Y 587.324,Z 136.822,A -85,B 0,C 180,E1 -1585.653,E2 -1585.653} C_VEL
LIN {X 0,Y 587.303,Z 136.822,A -85,B 0,C 180,E1 -1588.228,E2 -1588.228} C_VEL
LIN {X 0,Y 587.326,Z 136.826,A -85,B 0,C 180,E1 -1590.868,E2 -1590.868} C_VEL
LIN {X 0,Y 587.282,Z 136.825,A -85,B 0,C 180,E1 -1593.831,E2 -1593.831} C_VEL
LIN {X 0,Y 587.282,Z 136.831,A -85,B 0,C 180,E1 -1596.739,E2 -1596.739} C_VEL
LIN {X 0,Y 587.293,Z 136.824,A -85,B 0,C 180,E1 -1599.694,E2 -1599.694} C_VEL
LIN {X 0,Y 587.268,Z 136.826,A -85,B 0,C 180,E1 -1601.871,E2 -1601.871} C_VEL
LIN {X 0,Y 587.285,Z 136.825,A -85,B 0,C 180,E1 -1604.023,E2 -1604.023} C_VEL
LIN {X 0,Y 587.275,Z 136.835,A -85,B 0,C 180,E1 -1606.857,E2 -1606.857} C_VEL
LIN {X 0,Y 587.322,Z 136.826,A -85,B 0,C 180,E1 -1608.962,E2 -1608.962} C_VEL
LIN {X 0,Y 587.297,Z 136.823,A -85,B 0,C 180,E1 -1611.743,E2 -1611.743} C_VEL
LIN {X 0,Y 587.337,Z 136.826,A -85,B 0,C 180,E1 -1614.507,E2 -1614.507} C_VEL
LIN {X 0,Y 587.329,Z 136.82,A -85,B 0,C 180,E1 -1617.256,E2 -1617.256} C_VEL
LIN {X 0,Y 587.343,Z 136.819,A -85,B 0,C 180,E1 -1620,E2 -1620} C_VEL
LIN {X 0,Y 587.355,Z 136.822,A -85,B 0,C 180,E1 -1622.743,E2 -1622.743} C_VEL
LIN {X 0,Y 587.307,Z 136.822,A -85,B 0,C 180,E1 -1625.493,E2 -1625.493} C_VEL
LIN {X 0,Y 587.287,Z 136.824,A -85,B 0,C 180,E1 -1627.564,E2 -1627.564} C_VEL
LIN {X 0,Y 587.306,Z 136.831,A -85,B 0,C 180,E1 -1630.34,E2 -1630.34} C_VEL
LIN {X 0,Y 587.278,Z 136.826,A -85,B 0,C 180,E1 -1633.142,E2 -1633.142} C_VEL
LIN {X 0,Y 587.284,Z 136.825,A -85,B 0,C 180,E1 -1635.329,E2 -1635.329} C_VEL
LIN {X 0,Y 587.265,Z 136.835,A -85,B 0,C 180,E1 -1638.128,E2 -1638.128} C_VEL
LIN {X 0,Y 587.269,Z 136.832,A -85,B 0,C 180,E1 -1638.317,E2 -1638.317} C_VEL
LIN {X 0,Y 586.632,Z 136.908,A -85,B 0,C 180,E1 -1638.889,E2 -1638.889} C_VEL
LIN {X 0,Y 583.819,Z 137.26,A -85,B 0,C 180,E1 -1639.818,E2 -1639.818} C_VEL
LIN {X 0,Y 581.415,Z 137.561,A -85,B 0,C 180,E1 -1640.565,E2 -1640.565} C_VEL
LIN {X 0,Y 580.361,Z 137.688,A -85,B 0,C 180,E1 -1641.142,E2 -1641.142} C_VEL
LIN {X 0,Y 580.264,Z 137.7,A -85,B 0,C 180,E1 -1641.337,E2 -1641.337} C_VEL
LIN {X 0,Y 580.267,Z 137.706,A -85,B 0,C 180,E1 -1644.317,E2 -1644.317} C_VEL
LIN {X 0,Y 580.224,Z 137.707,A -85,B 0,C 180,E1 -1646.626,E2 -1646.626} C_VEL
LIN {X 0,Y 580.238,Z 137.704,A -85,B 0,C 180,E1 -1649.301,E2 -1649.301} C_VEL
LIN {X 0,Y 580.268,Z 137.708,A -85,B 0,C 180,E1 -1652.202,E2 -1652.202} C_VEL
LIN {X 0,Y 580.318,Z 137.877,A -85,B 0,C 180,E1 -1653.59,E2 -1653.59} C_VEL
LIN {X 0,Y 580.621,Z 142.676,A -85,B 0,C 180,E1 -1654.409,E2 -1654.409} C_VEL
LIN {X 0,Y 580.468,Z 159.773,A -85,B 0,C 180,E1 -1657.255,E2 -1657.255} C_VEL
LIN {X 0,Y 580.333,Z 177.122,A -85,B 0,C 180,E1 -1660.104,E2 -1660.104} C_VEL
LIN {X 0,Y 580.355,Z 179.04,A -85,B 0,C 180,E1 -1660.373,E2 -1660.373} C_VEL
LIN {X 0,Y 580.936,Z 183.597,A -85,B 0,C 180,E1 -1660.468,E2 -1660.468} C_VEL
LIN {X 0,Y 580.819,Z 286.555,A -85,B 0,C 180,E1 -1661.764,E2 -1661.764} C_VEL
LIN {X 0,Y 580.728,Z 299.684,A -85,B 0,C 180,E1 -1662.078,E2 -1662.078} C_VEL
LIN {X 0,Y 580.674,Z 309.598,A -85,B 0,C 180,E1 -1662.416,E2 -1662.416} C_VEL
LIN {X 0,Y 580.558,Z 320.909,A -85,B 0,C 180,E1 -1662.917,E2 -1662.917} C_VEL
LIN {X 0,Y 580.478,Z 332.361,A -85,B 0,C 180,E1 -1663.568,E2 -1663.568} C_VEL
LIN {X 0,Y 580.39,Z 343.846,A -85,B 0,C 180,E1 -1664.405,E2 -1664.405} C_VEL
LIN {X 0,Y 580.291,Z 353.245,A -85,B 0,C 180,E1 -1665.256,E2 -1665.256} C_VEL
LIN {X 0,Y 580.21,Z 360.939,A -85,B 0,C 180,E1 -1666.097,E2 -1666.097} C_VEL
LIN {X 0,Y 580.176,Z 368.671,A -85,B 0,C 180,E1 -1667.119,E2 -1667.119} C_VEL
LIN {X 0,Y 580.146,Z 375.321,A -85,B 0,C 180,E1 -1668.221,E2 -1668.221} C_VEL
LIN {X 0,Y 580.098,Z 381.115,A -85,B 0,C 180,E1 -1669.471,E2 -1669.471} C_VEL
LIN {X 0,Y 580.044,Z 384.623,A -85,B 0,C 180,E1 -1670.471,E2 -1670.471} C_VEL
LIN {X 0,Y 580.06,Z 386.015,A -85,B 0,C 180,E1 -1670.949,E2 -1670.949} C_VEL
LIN {X 0,Y 580.018,Z 388.209,A -85,B 0,C 180,E1 -1671.961,E2 -1671.961} C_VEL
LIN {X 0,Y 580.025,Z 389.622,A -85,B 0,C 180,E1 -1673.101,E2 -1673.101} C_VEL
LIN {X 0,Y 580.038,Z 389.9,A -85,B 0,C 180,E1 -1674.439,E2 -1674.439} C_VEL
LIN {X 0,Y 580.045,Z 389.118,A -85,B 0,C 180,E1 -1675.477,E2 -1675.477} C_VEL
LIN {X 0,Y 580.055,Z 387,A -85,B 0,C 180,E1 -1676.72,E2 -1676.72} C_VEL
LIN {X 0,Y 580.074,Z 383.43,A -85,B 0,C 180,E1 -1678.005,E2 -1678.005} C_VEL
LIN {X 0,Y 580.114,Z 378.005,A -85,B 0,C 180,E1 -1679.333,E2 -1679.333} C_VEL
LIN {X 0,Y 580.146,Z 373.344,A -85,B 0,C 180,E1 -1680.221,E2 -1680.221} C_VEL
LIN {X 0,Y 580.176,Z 366.923,A -85,B 0,C 180,E1 -1681.217,E2 -1681.217} C_VEL
LIN {X 0,Y 580.231,Z 359.578,A -85,B 0,C 180,E1 -1682.153,E2 -1682.153} C_VEL
LIN {X 0,Y 580.317,Z 350.681,A -85,B 0,C 180,E1 -1683.088,E2 -1683.088} C_VEL
LIN {X 0,Y 580.373,Z 339.817,A -85,B 0,C 180,E1 -1684.003,E2 -1684.003} C_VEL
LIN {X 0,Y 580.484,Z 330.409,A -85,B 0,C 180,E1 -1684.642,E2 -1684.642} C_VEL
LIN {X 0,Y 580.571,Z 320.047,A -85,B 0,C 180,E1 -1685.216,E2 -1685.216} C_VEL
LIN {X 0,Y 580.645,Z 308.957,A -85,B 0,C 180,E1 -1685.7,E2 -1685.7} C_VEL
LIN {X 0,Y 580.745,Z 295.972,A -85,B 0,C 180,E1 -1686.12,E2 -1686.12} C_VEL
LIN {X 0,Y 580.823,Z 282.851,A -85,B 0,C 180,E1 -1686.384,E2 -1686.384} C_VEL
LIN {X 0,Y 580.817,Z 182.165,A -85,B 0,C 180,E1 -1687.643,E2 -1687.643} C_VEL
LIN {X 0,Y 580.386,Z 178.985,A -85,B 0,C 180,E1 -1687.719,E2 -1687.719} C_VEL
LIN {X 0,Y 580.421,Z 161.526,A -85,B 0,C 180,E1 -1690.546,E2 -1690.546} C_VEL
LIN {X 0,Y 580.603,Z 143.917,A -85,B 0,C 180,E1 -1693.474,E2 -1693.474} C_VEL
LIN {X 0,Y 580.389,Z 138.161,A -85,B 0,C 180,E1 -1694.461,E2 -1694.461} C_VEL
LIN {X 0,Y 580.31,Z 137.719,A -85,B 0,C 180,E1 -1694.639,E2 -1694.639} C_VEL
LIN {X 0,Y 580.303,Z 137.697,A -85,B 0,C 180,E1 -1697.41,E2 -1697.41} C_VEL
LIN {X 0,Y 580.27,Z 137.704,A -85,B 0,C 180,E1 -1700.239,E2 -1700.239} C_VEL
LIN {X 0,Y 580.325,Z 137.695,A -85,B 0,C 180,E1 -1702.345,E2 -1702.345} C_VEL
LIN {X 0,Y 580.331,Z 137.691,A -85,B 0,C 180,E1 -1705.138,E2 -1705.138} C_VEL
LIN {X 0,Y 580.332,Z 137.699,A -85,B 0,C 180,E1 -1707.919,E2 -1707.919} C_VEL
LIN {X 0,Y 580.356,Z 137.688,A -85,B 0,C 180,E1 -1710.695,E2 -1710.695} C_VEL
LIN {X 0,Y 580.284,Z 137.703,A -85,B 0,C 180,E1 -1713.472,E2 -1713.472} C_VEL
LIN {X 0,Y 580.32,Z 137.701,A -85,B 0,C 180,E1 -1715.56,E2 -1715.56} C_VEL
LIN {X 0,Y 580.322,Z 137.701,A -85,B 0,C 180,E1 -1717.656,E2 -1717.656} C_VEL
LIN {X 0,Y 580.295,Z 137.695,A -85,B 0,C 180,E1 -1720.467,E2 -1720.467} C_VEL
LIN {X 0,Y 580.299,Z 137.695,A -85,B 0,C 180,E1 -1722.592,E2 -1722.592} C_VEL
LIN {X 0,Y 580.284,Z 137.698,A -85,B 0,C 180,E1 -1724.735,E2 -1724.735} C_VEL
LIN {X 0,Y 580.289,Z 137.702,A -85,B 0,C 180,E1 -1727.625,E2 -1727.625} C_VEL
LIN {X 0,Y 580.285,Z 137.699,A -85,B 0,C 180,E1 -1729.823,E2 -1729.823} C_VEL
LIN {X 0,Y 580.268,Z 137.699,A -85,B 0,C 180,E1 -1732.053,E2 -1732.053} C_VEL
LIN {X 0,Y 580.301,Z 137.703,A -85,B 0,C 180,E1 -1735.08,E2 -1735.08} C_VEL
LIN {X 0,Y 580.298,Z 137.695,A -85,B 0,C 180,E1 -1738.186,E2 -1738.186} C_VEL
LIN {X 0,Y 580.271,Z 137.702,A -85,B 0,C 180,E1 -1740.693,E2 -1740.693} C_VEL
LIN {X 0,Y 580.282,Z 137.702,A -85,B 0,C 180,E1 -1743.314,E2 -1743.314} C_VEL
LIN {X 0,Y 580.243,Z 137.702,A -85,B 0,C 180,E1 -1745.756,E2 -1745.756} C_VEL
LIN {X 0,Y 580.285,Z 137.697,A -85,B 0,C 180,E1 -1748.147,E2 -1748.147} C_VEL
LIN {X 0,Y 580.293,Z 137.706,A -85,B 0,C 180,E1 -1750.844,E2 -1750.844} C_VEL
LIN {X 0,Y 580.267,Z 137.699,A -85,B 0,C 180,E1 -1753.659,E2 -1753.659} C_VEL
LIN {X 0,Y 580.265,Z 137.707,A -85,B 0,C 180,E1 -1756.611,E2 -1756.611} C_VEL
LIN {X 0,Y 580.293,Z 137.698,A -85,B 0,C 180,E1 -1759.157,E2 -1759.157} C_VEL
LIN {X 0,Y 580.284,Z 137.698,A -85,B 0,C 180,E1 -1761.928,E2 -1761.928} C_VEL
LIN {X 0,Y 580.247,Z 137.71,A -85,B 0,C 180,E1 -1764.453,E2 -1764.453} C_VEL
LIN {X 0,Y 580.286,Z 137.699,A -85,B 0,C 180,E1 -1766.975,E2 -1766.975} C_VEL
LIN {X 0,Y 580.288,Z 137.696,A -85,B 0,C 180,E1 -1769.425,E2 -1769.425} C_VEL
LIN {X 0,Y 580.255,Z 137.706,A -85,B 0,C 180,E1 -1772.149,E2 -1772.149} C_VEL
LIN {X 0,Y 580.319,Z 137.692,A -85,B 0,C 180,E1 -1775.27,E2 -1775.27} C_VEL
LIN {X 0,Y 580.251,Z 137.706,A -85,B 0,C 180,E1 -1777.947,E2 -1777.947} C_VEL
LIN {X 0,Y 580.295,Z 137.696,A -85,B 0,C 180,E1 -1780.85,E2 -1780.85} C_VEL
LIN {X 0,Y 580.252,Z 137.706,A -85,B 0,C 180,E1 -1783.825,E2 -1783.825} C_VEL
LIN {X 0,Y 580.309,Z 137.702,A -85,B 0,C 180,E1 -1785.983,E2 -1785.983} C_VEL
LIN {X 0,Y 580.304,Z 137.694,A -85,B 0,C 180,E1 -1788.827,E2 -1788.827} C_VEL
LIN {X 0,Y 580.304,Z 137.699,A -85,B 0,C 180,E1 -1791.644,E2 -1791.644} C_VEL
LIN {X 0,Y 580.296,Z 137.697,A -85,B 0,C 180,E1 -1794.44,E2 -1794.44} C_VEL
LIN {X 0,Y 580.323,Z 137.693,A -85,B 0,C 180,E1 -1797.224,E2 -1797.224} C_VEL
LIN {X 0,Y 580.341,Z 137.696,A -85,B 0,C 180,E1 -1800,E2 -1800} C_VEL
LIN {X 0,Y 580.31,Z 137.693,A -85,B 0,C 180,E1 -1802.777,E2 -1802.777} C_VEL
LIN {X 0,Y 580.309,Z 137.702,A -85,B 0,C 180,E1 -1805.56,E2 -1805.56} C_VEL
LIN {X 0,Y 580.288,Z 137.697,A -85,B 0,C 180,E1 -1808.357,E2 -1808.357} C_VEL
LIN {X 0,Y 580.301,Z 137.699,A -85,B 0,C 180,E1 -1811.191,E2 -1811.191} C_VEL
LIN {X 0,Y 580.267,Z 137.699,A -85,B 0,C 180,E1 -1814.32,E2 -1814.32} C_VEL
LIN {X 0,Y 580.267,Z 137.701,A -85,B 0,C 180,E1 -1816.899,E2 -1816.899} C_VEL
LIN {X 0,Y 580.27,Z 137.701,A -85,B 0,C 180,E1 -1819.824,E2 -1819.824} C_VEL
LIN {X 0,Y 580.277,Z 137.7,A -85,B 0,C 180,E1 -1822.803,E2 -1822.803} C_VEL
LIN {X 0,Y 580.244,Z 137.703,A -85,B 0,C 180,E1 -1825.852,E2 -1825.852} C_VEL
LIN {X 0,Y 580.228,Z 137.704,A -85,B 0,C 180,E1 -1828.19,E2 -1828.19} C_VEL
LIN {X 0,Y 580.241,Z 137.705,A -85,B 0,C 180,E1 -1830.687,E2 -1830.687} C_VEL
LIN {X 0,Y 580.248,Z 137.707,A -85,B 0,C 180,E1 -1833.308,E2 -1833.308} C_VEL
LIN {X 0,Y 580.216,Z 137.706,A -85,B 0,C 180,E1 -1835.752,E2 -1835.752} C_VEL
LIN {X 0,Y 580.273,Z 137.698,A -85,B 0,C 180,E1 -1838.148,E2 -1838.148} C_VEL
LIN {X 0,Y 580.239,Z 137.712,A -85,B 0,C 180,E1 -1840.849,E2 -1840.849} C_VEL
LIN {X 0,Y 580.226,Z 137.704,A -85,B 0,C 180,E1 -1843.663,E2 -1843.663} C_VEL
LIN {X 0,Y 580.225,Z 137.711,A -85,B 0,C 180,E1 -1846.615,E2 -1846.615} C_VEL
LIN {X 0,Y 580.239,Z 137.705,A -85,B 0,C 180,E1 -1849.151,E2 -1849.151} C_VEL
LIN {X 0,Y 580.234,Z 137.704,A -85,B 0,C 180,E1 -1851.935,E2 -1851.935} C_VEL
LIN {X 0,Y 580.205,Z 137.714,A -85,B 0,C 180,E1 -1854.449,E2 -1854.449} C_VEL
LIN {X 0,Y 580.238,Z 137.706,A -85,B 0,C 180,E1 -1856.971,E2 -1856.971} C_VEL
LIN {X 0,Y 580.25,Z 137.702,A -85,B 0,C 180,E1 -1859.422,E2 -1859.422} C_VEL
LIN {X 0,Y 580.23,Z 137.71,A -85,B 0,C 180,E1 -1862.155,E2 -1862.155} C_VEL
LIN {X 0,Y 580.245,Z 137.706,A -85,B 0,C 180,E1 -1864.917,E2 -1864.917} C_VEL
LIN {X 0,Y 580.296,Z 137.871,A -85,B 0,C 180,E1 -1867.714,E2 -1867.714} C_VEL
LIN {X 0,Y 580.839,Z 141.714,A -85,B 0,C 180,E1 -1868.343,E2 -1868.343} C_VEL
LIN {X 0,Y 580.644,Z 159.987,A -85,B 0,C 180,E1 -1871.108,E2 -1871.108} C_VEL
LIN {X 0,Y 580.51,Z 176.977,A -85,B 0,C 180,E1 -1873.651,E2 -1873.651} C_VEL
LIN {X 0,Y 580.402,Z 195.241,A -85,B 0,C 180,E1 -1876.319,E2 -1876.319} C_VEL
LIN {X 0,Y 580.945,Z 200.465,A -85,B 0,C 180,E1 -1876.422,E2 -1876.422} C_VEL
LIN {X 0,Y 580.806,Z 302.918,A -85,B 0,C 180,E1 -1877.708,E2 -1877.708} C_VEL
LIN {X 0,Y 580.744,Z 316.2,A -85,B 0,C 180,E1 -1878.017,E2 -1878.017} C_VEL
LIN {X 0,Y 580.642,Z 329.481,A -85,B 0,C 180,E1 -1878.48,E2 -1878.48} C_VEL
LIN {X 0,Y 580.563,Z 340.617,A -85,B 0,C 180,E1 -1879.008,E2 -1879.008} C_VEL
LIN {X 0,Y 580.448,Z 352.192,A -85,B 0,C 180,E1 -1879.712,E2 -1879.712} C_VEL
LIN {X 0,Y 580.345,Z 362.594,A -85,B 0,C 180,E1 -1880.502,E2 -1880.502} C_VEL
LIN {X 0,Y 580.267,Z 371.107,A -85,B 0,C 180,E1 -1881.292,E2 -1881.292} C_VEL
LIN {X 0,Y 580.222,Z 378.955,A -85,B 0,C 180,E1 -1882.168,E2 -1882.168} C_VEL
LIN {X 0,Y 580.154,Z 386.648,A -85,B 0,C 180,E1 -1883.221,E2 -1883.221} C_VEL
LIN {X 0,Y 580.139,Z 393.677,A -85,B 0,C 180,E1 -1884.438,E2 -1884.438} C_VEL
LIN {X 0,Y 580.108,Z 398.369,A -85,B 0,C 180,E1 -1885.483,E2 -1885.483} C_VEL
LIN {X 0,Y 580.123,Z 401.955,A -85,B 0,C 180,E1 -1886.527,E2 -1886.527} C_VEL
LIN {X 0,Y 580.043,Z 403.807,A -85,B 0,C 180,E1 -1887.221,E2 -1887.221} C_VEL
LIN {X 0,Y 580.04,Z 405.197,A -85,B 0,C 180,E1 -1887.916,E2 -1887.916} C_VEL
LIN {X 0,Y 580.04,Z 406.784,A -85,B 0,C 180,E1 -1889.305,E2 -1889.305} C_VEL
LIN {X 0,Y 580.037,Z 407,A -85,B 0,C 180,E1 -1889.999,E2 -1889.999} C_VEL
LIN {X 0,Y 580.047,Z 406.187,A -85,B 0,C 180,E1 -1891.388,E2 -1891.388} C_VEL
LIN {X 0,Y 580.04,Z 405.201,A -85,B 0,C 180,E1 -1892.082,E2 -1892.082} C_VEL
LIN {X 0,Y 580.043,Z 403.812,A -85,B 0,C 180,E1 -1892.777,E2 -1892.777} C_VEL
LIN {X 0,Y 580.11,Z 400.898,A -85,B 0,C 180,E1 -1893.82,E2 -1893.82} C_VEL
LIN {X 0,Y 580.053,Z 396.952,A -85,B 0,C 180,E1 -1894.864,E2 -1894.864} C_VEL
LIN {X 0,Y 580.139,Z 390.881,A -85,B 0,C 180,E1 -1896.084,E2 -1896.084} C_VEL
LIN {X 0,Y 580.183,Z 384.243,A -85,B 0,C 180,E1 -1897.132,E2 -1897.132} C_VEL
LIN {X 0,Y 580.25,Z 375.998,A -85,B 0,C 180,E1 -1898.181,E2 -1898.181} C_VEL
LIN {X 0,Y 580.307,Z 367.548,A -85,B 0,C 180,E1 -1899.057,E2 -1899.057} C_VEL
LIN {X 0,Y 580.426,Z 357.11,A -85,B 0,C 180,E1 -1899.935,E2 -1899.935} C_VEL
LIN {X 0,Y 580.516,Z 346.769,A -85,B 0,C 180,E1 -1900.638,E2 -1900.638} C_VEL
LIN {X 0,Y 580.596,Z 335.246,A -85,B 0,C 180,E1 -1901.264,E2 -1901.264} C_VEL
LIN {X 0,Y 580.679,Z 322.499,A -85,B 0,C 180,E1 -1901.784,E2 -1901.784} C_VEL
LIN {X 0,Y 580.784,Z 309.471,A -85,B 0,C 180,E1 -1902.158,E2 -1902.158} C_VEL
LIN {X 0,Y 580.831,Z 297.152,A -85,B 0,C 180,E1 -1902.379,E2 -1902.379} C_VEL
LIN {X 0,Y 580.905,Z 198.796,A -85,B 0,C 180,E1 -1903.6,E2 -1903.6} C_VEL
LIN {X 0,Y 580.387,Z 195.264,A -85,B 0,C 180,E1 -1903.68,E2 -1903.68} C_VEL
LIN {X 0,Y 580.508,Z 176.987,A -85,B 0,C 180,E1 -1906.347,E2 -1906.347} C_VEL
LIN {X 0,Y 580.641,Z 159.997,A -85,B 0,C 180,E1 -1908.891,E2 -1908.891} C_VEL
LIN {X 0,Y 580.805,Z 143.018,A -85,B 0,C 180,E1 -1911.452,E2 -1911.452} C_VEL
LIN {X 0,Y 580.538,Z 139.203,A -85,B 0,C 180,E1 -1912.041,E2 -1912.041} C_VEL
LIN {X 0,Y 580.266,Z 137.757,A -85,B 0,C 180,E1 -1912.333,E2 -1912.333} C_VEL
LIN {X 0,Y 580.276,Z 137.702,A -85,B 0,C 180,E1 -1915.08,E2 -1915.08} C_VEL
LIN {X 0,Y 580.232,Z 137.71,A -85,B 0,C 180,E1 -1917.846,E2 -1917.846} C_VEL
LIN {X 0,Y 580.238,Z 137.703,A -85,B 0,C 180,E1 -1920.686,E2 -1920.686} C_VEL
LIN {X 0,Y 580.273,Z 137.705,A -85,B 0,C 180,E1 -1923.311,E2 -1923.311} C_VEL
LIN {X 0,Y 580.216,Z 137.711,A -85,B 0,C 180,E1 -1925.752,E2 -1925.752} C_VEL
LIN {X 0,Y 580.228,Z 137.704,A -85,B 0,C 180,E1 -1928.149,E2 -1928.149} C_VEL
LIN {X 0,Y 580.248,Z 137.704,A -85,B 0,C 180,E1 -1930.846,E2 -1930.846} C_VEL
LIN {X 0,Y 580.219,Z 137.709,A -85,B 0,C 180,E1 -1933.662,E2 -1933.662} C_VEL
LIN {X 0,Y 580.223,Z 137.705,A -85,B 0,C 180,E1 -1936.613,E2 -1936.613} C_VEL
LIN {X 0,Y 580.267,Z 137.701,A -85,B 0,C 180,E1 -1939.73,E2 -1939.73} C_VEL
LIN {X 0,Y 580.259,Z 137.702,A -85,B 0,C 180,E1 -1942.728,E2 -1942.728} C_VEL
LIN {X 0,Y 580.276,Z 137.702,A -85,B 0,C 180,E1 -1945.442,E2 -1945.442} C_VEL
LIN {X 0,Y 580.269,Z 137.698,A -85,B 0,C 180,E1 -1947.972,E2 -1947.972} C_VEL
LIN {X 0,Y 580.265,Z 137.709,A -85,B 0,C 180,E1 -1951.022,E2 -1951.022} C_VEL
LIN {X 0,Y 580.241,Z 137.703,A -85,B 0,C 180,E1 -1953.673,E2 -1953.673} C_VEL
LIN {X 0,Y 580.232,Z 137.705,A -85,B 0,C 180,E1 -1956.44,E2 -1956.44} C_VEL
LIN {X 0,Y 580.246,Z 137.703,A -85,B 0,C 180,E1 -1959.436,E2 -1959.436} C_VEL
LIN {X 0,Y 580.23,Z 137.704,A -85,B 0,C 180,E1 -1961.644,E2 -1961.644} C_VEL
LIN {X 0,Y 580.236,Z 137.702,A -85,B 0,C 180,E1 -1963.824,E2 -1963.824} C_VEL
LIN {X 0,Y 580.231,Z 137.712,A -85,B 0,C 180,E1 -1966.695,E2 -1966.695} C_VEL
LIN {X 0,Y 580.291,Z 137.704,A -85,B 0,C 180,E1 -1968.826,E2 -1968.826} C_VEL
LIN {X 0,Y 580.271,Z 137.698,A -85,B 0,C 180,E1 -1971.643,E2 -1971.643} C_VEL
LIN {X 0,Y 580.299,Z 137.701,A -85,B 0,C 180,E1 -1974.44,E2 -1974.44} C_VEL
LIN {X 0,Y 580.299,Z 137.696,A -85,B 0,C 180,E1 -1977.223,E2 -1977.223} C_VEL
LIN {X 0,Y 580.314,Z 137.695,A -85,B 0,C 180,E1 -1980,E2 -1980} C_VEL
LIN {X 0,Y 580.317,Z 137.698,A -85,B 0,C 180,E1 -1982.776,E2 -1982.776} C_VEL
LIN {X 0,Y 580.276,Z 137.698,A -85,B 0,C 180,E1 -1985.56,E2 -1985.56} C_VEL
LIN {X 0,Y 580.24,Z 137.703,A -85,B 0,C 180,E1 -1987.656,E2 -1987.656} C_VEL
LIN {X 0,Y 580.26,Z 137.709,A -85,B 0,C 180,E1 -1990.467,E2 -1990.467} C_VEL
LIN {X 0,Y 580.274,Z 137.704,A -85,B 0,C 180,E1 -1992.592,E2 -1992.592} C_VEL
LIN {X 0,Y 580.256,Z 137.701,A -85,B 0,C 180,E1 -1995.453,E2 -1995.453} C_VEL
LIN {X 0,Y 580.226,Z 137.713,A -85,B 0,C 180,E1 -1998.356,E2 -1998.356} C_VEL
LIN {X 0,Y 580.285,Z 137.697,A -85,B 0,C 180,E1 -2001.166,E2 -2001.166} C_VEL
LIN {X 0,Y 580.264,Z 137.7,A -85,B 0,C 180,E1 -2001.337,E2 -2001.337} C_VEL
LIN {X 0,Y 579.565,Z 137.794,A -85,B 0,C 180,E1 -2001.916,E2 -2001.916} C_VEL
LIN {X 0,Y 576.688,Z 138.148,A -85,B 0,C 180,E1 -2002.856,E2 -2002.856} C_VEL
LIN {X 0,Y 574.287,Z 138.447,A -85,B 0,C 180,E1 -2003.612,E2 -2003.612} C_VEL
LIN {X 0,Y 573.274,Z 138.579,A -85,B 0,C 180,E1 -2004.196,E2 -2004.196} C_VEL
LIN {X 0,Y 573.2,Z 138.581,A -85,B 0,C 180,E1 -2004.394,E2 -2004.394} C_VEL
LIN {X 0,Y 573.171,Z 138.584,A -85,B 0,C 180,E1 -2006.98,E2 -2006.98} C_VEL
LIN {X 0,Y 573.191,Z 138.583,A -85,B 0,C 180,E1 -2009.481,E2 -2009.481} C_VEL
LIN {X 0,Y 573.221,Z 138.586,A -85,B 0,C 180,E1 -2012.226,E2 -2012.226} C_VEL
LIN {X 0,Y 573.272,Z 138.664,A -85,B 0,C 180,E1 -2013.482,E2 -2013.482} C_VEL
LIN {X 0,Y 573.649,Z 142.057,A -85,B 0,C 180,E1 -2014.09,E2 -2014.09} C_VEL
LIN {X 0,Y 573.511,Z 158.922,A -85,B 0,C 180,E1 -2016.903,E2 -2016.903} C_VEL
LIN {X 0,Y 573.319,Z 176.512,A -85,B 0,C 180,E1 -2019.829,E2 -2019.829} C_VEL
LIN {X 0,Y 573.353,Z 178.984,A -85,B 0,C 180,E1 -2020.199,E2 -2020.199} C_VEL
LIN {X 0,Y 573.944,Z 183.04,A -85,B 0,C 180,E1 -2020.292,E2 -2020.292} C_VEL
LIN {X 0,Y 573.893,Z 286.604,A -85,B 0,C 180,E1 -2021.615,E2 -2021.615} C_VEL
LIN {X 0,Y 573.772,Z 299.283,A -85,B 0,C 180,E1 -2021.92,E2 -2021.92} C_VEL
LIN {X 0,Y 573.698,Z 310.423,A -85,B 0,C 180,E1 -2022.306,E2 -2022.306} C_VEL
LIN {X 0,Y 573.574,Z 321.024,A -85,B 0,C 180,E1 -2022.786,E2 -2022.786} C_VEL
LIN {X 0,Y 573.491,Z 332.085,A -85,B 0,C 180,E1 -2023.422,E2 -2023.422} C_VEL
LIN {X 0,Y 573.344,Z 343.266,A -85,B 0,C 180,E1 -2024.237,E2 -2024.237} C_VEL
LIN {X 0,Y 573.246,Z 352.078,A -85,B 0,C 180,E1 -2025.03,E2 -2025.03} C_VEL
LIN {X 0,Y 573.147,Z 359.636,A -85,B 0,C 180,E1 -2025.844,E2 -2025.844} C_VEL
LIN {X 0,Y 573.113,Z 365.83,A -85,B 0,C 180,E1 -2026.631,E2 -2026.631} C_VEL
LIN {X 0,Y 573.061,Z 372.107,A -85,B 0,C 180,E1 -2027.585,E2 -2027.585} C_VEL
LIN {X 0,Y 573.041,Z 377.2,A -85,B 0,C 180,E1 -2028.528,E2 -2028.528} C_VEL
LIN {X 0,Y 573.004,Z 381.449,A -85,B 0,C 180,E1 -2029.503,E2 -2029.503} C_VEL
LIN {X 0,Y 572.946,Z 385.142,A -85,B 0,C 180,E1 -2030.604,E2 -2030.604} C_VEL
LIN {X 0,Y 572.932,Z 387.805,A -85,B 0,C 180,E1 -2031.727,E2 -2031.727} C_VEL
LIN {X 0,Y 572.945,Z 389.601,A -85,B 0,C 180,E1 -2033.056,E2 -2033.056} C_VEL
LIN {X 0,Y 572.918,Z 390,A -85,B 0,C 180,E1 -2034.059,E2 -2034.059} C_VEL
LIN {X 0,Y 572.956,Z 389.377,A -85,B 0,C 180,E1 -2035.268,E2 -2035.268} C_VEL
LIN {X 0,Y 572.958,Z 387.476,A -85,B 0,C 180,E1 -2036.521,E2 -2036.521} C_VEL
LIN {X 0,Y 572.985,Z 384.169,A -85,B 0,C 180,E1 -2037.814,E2 -2037.814} C_VEL
LIN {X 0,Y 573.013,Z 379.148,A -85,B 0,C 180,E1 -2039.153,E2 -2039.153} C_VEL
LIN {X 0,Y 573.078,Z 373.854,A -85,B 0,C 180,E1 -2040.208,E2 -2040.208} C_VEL
LIN {X 0,Y 573.114,Z 367.449,A -85,B 0,C 180,E1 -2041.23,E2 -2041.23} C_VEL
LIN {X 0,Y 573.156,Z 361.28,A -85,B 0,C 180,E1 -2042.049,E2 -2042.049} C_VEL
LIN {X 0,Y 573.226,Z 354.377,A -85,B 0,C 180,E1 -2042.827,E2 -2042.827} C_VEL
LIN {X 0,Y 573.313,Z 345.579,A -85,B 0,C 180,E1 -2043.655,E2 -2043.655} C_VEL
LIN {X 0,Y 573.424,Z 335.952,A -85,B 0,C 180,E1 -2044.405,E2 -2044.405} C_VEL
LIN {X 0,Y 573.585,Z 323.517,A -85,B 0,C 180,E1 -2045.177,E2 -2045.177} C_VEL
LIN {X 0,Y 573.663,Z 311.979,A -85,B 0,C 180,E1 -2045.722,E2 -2045.722} C_VEL
LIN {X 0,Y 573.77,Z 301.199,A -85,B 0,C 180,E1 -2046.112,E2 -2046.112} C_VEL
LIN {X 0,Y 573.869,Z 289.096,A -85,B 0,C 180,E1 -2046.427,E2 -2046.427} C_VEL
LIN {X 0,Y 573.903,Z 270.36,A -85,B 0,C 180,E1 -2046.699,E2 -2046.699} C_VEL
LIN {X 0,Y 573.999,Z 183.589,A -85,B 0,C 180,E1 -2047.789,E2 -2047.789} C_VEL
LIN {X 0,Y 573.354,Z 179.122,A -85,B 0,C 180,E1 -2047.882,E2 -2047.882} C_VEL
LIN {X 0,Y 573.302,Z 175.535,A -85,B 0,C 180,E1 -2048.423,E2 -2048.423} C_VEL
LIN {X 0,Y 573.475,Z 158.622,A -85,B 0,C 180,E1 -2051.239,E2 -2051.239} C_VEL
LIN {X 0,Y 573.649,Z 141.243,A -85,B 0,C 180,E1 -2054.182,E2 -2054.182} C_VEL
LIN {X 0,Y 573.297,Z 138.65,A -85,B 0,C 180,E1 -2054.674,E2 -2054.674} C_VEL
LIN {X 0,Y 573.262,Z 138.573,A -85,B 0,C 180,E1 -2057.252,E2 -2057.252} C_VEL
LIN {X 0,Y 573.266,Z 138.574,A -85,B 0,C 180,E1 -2059.404,E2 -2059.404} C_VEL
LIN {X 0,Y 573.277,Z 138.574,A -85,B 0,C 180,E1 -2062.251,E2 -2062.251} C_VEL
LIN {X 0,Y 573.303,Z 138.567,A -85,B 0,C 180,E1 -2065.078,E2 -2065.078} C_VEL
LIN {X 0,Y 573.303,Z 138.575,A -85,B 0,C 180,E1 -2067.893,E2 -2067.893} C_VEL
LIN {X 0,Y 573.327,Z 138.563,A -85,B 0,C 180,E1 -2070.703,E2 -2070.703} C_VEL
LIN {X 0,Y 573.235,Z 138.582,A -85,B 0,C 180,E1 -2073.515,E2 -2073.515} C_VEL
LIN {X 0,Y 573.287,Z 138.579,A -85,B 0,C 180,E1 -2075.629,E2 -2075.629} C_VEL
LIN {X 0,Y 573.27,Z 138.577,A -85,B 0,C 180,E1 -2077.751,E2 -2077.751} C_VEL
LIN {X 0,Y 573.263,Z 138.571,A -85,B 0,C 180,E1 -2080.597,E2 -2080.597} C_VEL
LIN {X 0,Y 573.259,Z 138.572,A -85,B 0,C 180,E1 -2082.749,E2 -2082.749} C_VEL
LIN {X 0,Y 573.232,Z 138.578,A -85,B 0,C 180,E1 -2084.92,E2 -2084.92} C_VEL
LIN {X 0,Y 573.239,Z 138.577,A -85,B 0,C 180,E1 -2087.849,E2 -2087.849} C_VEL
LIN {X 0,Y 573.24,Z 138.575,A -85,B 0,C 180,E1 -2090.078,E2 -2090.078} C_VEL
LIN {X 0,Y 573.233,Z 138.575,A -85,B 0,C 180,E1 -2092.338,E2 -2092.338} C_VEL
LIN {X 0,Y 573.245,Z 138.58,A -85,B 0,C 180,E1 -2095.411,E2 -2095.411} C_VEL
LIN {X 0,Y 573.25,Z 138.573,A -85,B 0,C 180,E1 -2098.029,E2 -2098.029} C_VEL
LIN {X 0,Y 573.221,Z 138.583,A -85,B 0,C 180,E1 -2100.881,E2 -2100.881} C_VEL
LIN {X 0,Y 573.24,Z 138.577,A -85,B 0,C 180,E1 -2103.521,E2 -2103.521} C_VEL
LIN {X 0,Y 573.213,Z 138.578,A -85,B 0,C 180,E1 -2106.052,E2 -2106.052} C_VEL
LIN {X 0,Y 573.239,Z 138.581,A -85,B 0,C 180,E1 -2108.702,E2 -2108.702} C_VEL
LIN {X 0,Y 573.226,Z 138.576,A -85,B 0,C 180,E1 -2111.593,E2 -2111.593} C_VEL
LIN {X 0,Y 573.227,Z 138.579,A -85,B 0,C 180,E1 -2114.334,E2 -2114.334} C_VEL
LIN {X 0,Y 573.231,Z 138.576,A -85,B 0,C 180,E1 -2117.36,E2 -2117.36} C_VEL
LIN {X 0,Y 573.236,Z 138.58,A -85,B 0,C 180,E1 -2120.392,E2 -2120.392} C_VEL
LIN {X 0,Y 573.228,Z 138.578,A -85,B 0,C 180,E1 -2123.076,E2 -2123.076} C_VEL
LIN {X 0,Y 573.261,Z 138.572,A -85,B 0,C 180,E1 -2125.671,E2 -2125.671} C_VEL
LIN {X 0,Y 573.234,Z 138.58,A -85,B 0,C 180,E1 -2128.185,E2 -2128.185} C_VEL
LIN {X 0,Y 573.257,Z 138.578,A -85,B 0,C 180,E1 -2130.634,E2 -2130.634} C_VEL
LIN {X 0,Y 573.212,Z 138.578,A -85,B 0,C 180,E1 -2133.513,E2 -2133.513} C_VEL
LIN {X 0,Y 573.225,Z 138.583,A -85,B 0,C 180,E1 -2136.135,E2 -2136.135} C_VEL
LIN {X 0,Y 573.245,Z 138.574,A -85,B 0,C 180,E1 -2139.174,E2 -2139.174} C_VEL
LIN {X 0,Y 573.205,Z 138.579,A -85,B 0,C 180,E1 -2141.411,E2 -2141.411} C_VEL
LIN {X 0,Y 573.226,Z 138.578,A -85,B 0,C 180,E1 -2143.621,E2 -2143.621} C_VEL
LIN {X 0,Y 573.255,Z 138.577,A -85,B 0,C 180,E1 -2145.807,E2 -2145.807} C_VEL
LIN {X 0,Y 573.262,Z 138.572,A -85,B 0,C 180,E1 -2148.746,E2 -2148.746} C_VEL
LIN {X 0,Y 573.247,Z 138.577,A -85,B 0,C 180,E1 -2151.54,E2 -2151.54} C_VEL
LIN {X 0,Y 573.266,Z 138.574,A -85,B 0,C 180,E1 -2154.372,E2 -2154.372} C_VEL
LIN {X 0,Y 573.299,Z 138.576,A -85,B 0,C 180,E1 -2157.893,E2 -2157.893} C_VEL
LIN {X 0,Y 573.31,Z 138.572,A -85,B 0,C 180,E1 -2160,E2 -2160} C_VEL
LIN {X 0,Y 573.28,Z 138.569,A -85,B 0,C 180,E1 -2162.811,E2 -2162.811} C_VEL
LIN {X 0,Y 573.274,Z 138.579,A -85,B 0,C 180,E1 -2165.629,E2 -2165.629} C_VEL
LIN {X 0,Y 573.233,Z 138.575,A -85,B 0,C 180,E1 -2168.461,E2 -2168.461} C_VEL
LIN {X 0,Y 573.272,Z 138.576,A -85,B 0,C 180,E1 -2171.312,E2 -2171.312} C_VEL
LIN {X 0,Y 573.226,Z 138.576,A -85,B 0,C 180,E1 -2174.402,E2 -2174.402} C_VEL
LIN {X 0,Y 573.237,Z 138.58,A -85,B 0,C 180,E1 -2177.113,E2 -2177.113} C_VEL
LIN {X 0,Y 573.225,Z 138.577,A -85,B 0,C 180,E1 -2180.078,E2 -2180.078} C_VEL
LIN {X 0,Y 573.215,Z 138.577,A -85,B 0,C 180,E1 -2182.339,E2 -2182.339} C_VEL
LIN {X 0,Y 573.205,Z 138.585,A -85,B 0,C 180,E1 -2185.413,E2 -2185.413} C_VEL
LIN {X 0,Y 573.196,Z 138.58,A -85,B 0,C 180,E1 -2188.018,E2 -2188.018} C_VEL
LIN {X 0,Y 573.203,Z 138.585,A -85,B 0,C 180,E1 -2190.878,E2 -2190.878} C_VEL
LIN {X 0,Y 573.216,Z 138.58,A -85,B 0,C 180,E1 -2193.517,E2 -2193.517} C_VEL
LIN {X 0,Y 573.182,Z 138.581,A -85,B 0,C 180,E1 -2196.054,E2 -2196.054} C_VEL
LIN {X 0,Y 573.228,Z 138.582,A -85,B 0,C 180,E1 -2198.703,E2 -2198.703} C_VEL
LIN {X 0,Y 573.186,Z 138.582,A -85,B 0,C 180,E1 -2201.588,E2 -2201.588} C_VEL
LIN {X 0,Y 573.203,Z 138.581,A -85,B 0,C 180,E1 -2204.337,E2 -2204.337} C_VEL
LIN {X 0,Y 573.207,Z 138.58,A -85,B 0,C 180,E1 -2207.363,E2 -2207.363} C_VEL
LIN {X 0,Y 573.216,Z 138.585,A -85,B 0,C 180,E1 -2210.572,E2 -2210.572} C_VEL
LIN {X 0,Y 573.215,Z 138.58,A -85,B 0,C 180,E1 -2213.074,E2 -2213.074} C_VEL
LIN {X 0,Y 573.17,Z 138.583,A -85,B 0,C 180,E1 -2215.664,E2 -2215.664} C_VEL
LIN {X 0,Y 573.207,Z 138.583,A -85,B 0,C 180,E1 -2218.182,E2 -2218.182} C_VEL
LIN {X 0,Y 573.213,Z 138.586,A -85,B 0,C 180,E1 -2220.631,E2 -2220.631} C_VEL
LIN {X 0,Y 573.197,Z 138.58,A -85,B 0,C 180,E1 -2223.516,E2 -2223.516} C_VEL
LIN {X 0,Y 573.192,Z 138.589,A -85,B 0,C 180,E1 -2226.132,E2 -2226.132} C_VEL
LIN {X 0,Y 573.251,Z 138.714,A -85,B 0,C 180,E1 -2227.567,E2 -2227.567} C_VEL
LIN {X 0,Y 573.892,Z 142.856,A -85,B 0,C 180,E1 -2228.256,E2 -2228.256} C_VEL
LIN {X 0,Y 573.661,Z 159.941,A -85,B 0,C 180,E1 -2230.869,E2 -2230.869} C_VEL
LIN {X 0,Y 573.523,Z 177.025,A -85,B 0,C 180,E1 -2233.453,E2 -2233.453} C_VEL
LIN {X 0,Y 573.399,Z 195.251,A -85,B 0,C 180,E1 -2236.149,E2 -2236.149} C_VEL
LIN {X 0,Y 574.046,Z 200.465,A -85,B 0,C 180,E1 -2236.255,E2 -2236.255} C_VEL
LIN {X 0,Y 573.891,Z 302.918,A -85,B 0,C 180,E1 -2237.557,E2 -2237.557} C_VEL
LIN {X 0,Y 573.793,Z 316.199,A -85,B 0,C 180,E1 -2237.869,E2 -2237.869} C_VEL
LIN {X 0,Y 573.678,Z 329.482,A -85,B 0,C 180,E1 -2238.338,E2 -2238.338} C_VEL
LIN {X 0,Y 573.59,Z 340.719,A -85,B 0,C 180,E1 -2238.879,E2 -2238.879} C_VEL
LIN {X 0,Y 573.44,Z 352.19,A -85,B 0,C 180,E1 -2239.585,E2 -2239.585} C_VEL
LIN {X 0,Y 573.333,Z 362.596,A -85,B 0,C 180,E1 -2240.385,E2 -2240.385} C_VEL
LIN {X 0,Y 573.239,Z 371.107,A -85,B 0,C 180,E1 -2241.184,E2 -2241.184} C_VEL
LIN {X 0,Y 573.161,Z 378.955,A -85,B 0,C 180,E1 -2242.07,E2 -2242.07} C_VEL
LIN {X 0,Y 573.073,Z 386.952,A -85,B 0,C 180,E1 -2243.185,E2 -2243.185} C_VEL
LIN {X 0,Y 573.071,Z 393.676,A -85,B 0,C 180,E1 -2244.369,E2 -2244.369} C_VEL
LIN {X 0,Y 573.029,Z 398.37,A -85,B 0,C 180,E1 -2245.427,E2 -2245.427} C_VEL
LIN {X 0,Y 573.022,Z 401.956,A -85,B 0,C 180,E1 -2246.484,E2 -2246.484} C_VEL
